Yaskawa INFORM job: test_long_tjr2.JBI

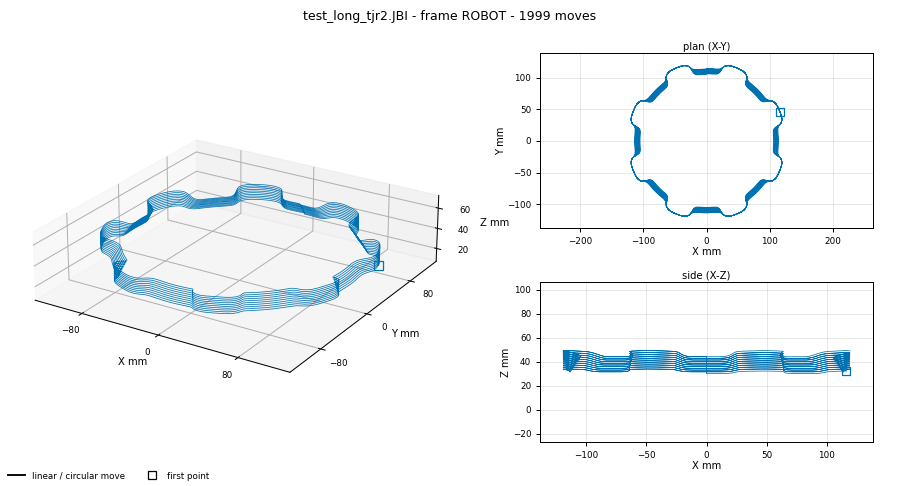
[picture p0: tool path of test_long_tjr2.JBI in frame ROBOT, 1999 of 2000 moves have a stored position in this frame; points joined in program order, loops and branches not executed]
version: 0
/JOB
//NAME test_long
//POS
///NPOS 48,0,0,2,0,0
///TOOL 1
///POSTYPE ROBOT
///RECTAN
///RCONF 1,0,0,0,0,0,0,0,0,0,0,0,0,0,0,0,0,0,0,0,0,0,0,0
C00000=117.720,41.900,32.250,-0.0000,-0.0000,1.0000
C00001=116.270,45.890,32.290,-0.0000,-0.0000,1.0000
C00002=114.660,49.770,32.290,-0.0000,-0.0000,1.0000
C00003=112.870,53.610,32.250,-0.0000,-0.0000,1.0000
C00004=110.690,57.360,32.180,0.0000,0.0000,1.0000
C00005=107.960,60.560,32.120,-0.0100,-0.0100,1.0000
C00006=105.150,62.790,32.030,-0.0300,-0.0400,1.0000
C00007=102.630,63.800,31.880,-0.0200,-0.0800,1.0000
C00008=100.220,64.240,31.550,-0.0200,-0.1500,0.9900
C00009=97.890,64.720,31.120,-0.0600,-0.2600,0.9600
C00010=95.560,65.770,30.680,-0.2000,-0.3600,0.9100
C00011=92.870,68.060,30.360,-0.3500,-0.3500,0.8700
C00012=89.340,72.130,30.220,-0.4000,-0.3400,0.8500
C00013=85.510,76.590,30.220,-0.3900,-0.3500,0.8500
C00014=81.180,81.180,30.220,-0.3700,-0.3700,0.8500
C00015=76.590,85.510,30.220,-0.3500,-0.3900,0.8500
C00016=72.130,89.340,30.220,-0.3400,-0.4000,0.8500
C00017=68.060,92.870,30.360,-0.3500,-0.3500,0.8700
C00018=65.770,95.560,30.680,-0.3600,-0.2000,0.9100
C00019=64.720,97.890,31.120,-0.2600,-0.0600,0.9600
C00020=64.240,100.220,31.550,-0.1500,-0.0200,0.9900
C00021=63.800,102.630,31.880,-0.0800,-0.0200,1.0000
C00022=62.790,105.150,32.030,-0.0400,-0.0300,1.0000
C00023=60.560,107.960,32.120,-0.0100,-0.0100,1.0000
C00024=57.360,110.690,32.180,0.0000,0.0000,1.0000
C00025=53.610,112.870,32.250,-0.0000,-0.0000,1.0000
C00026=49.770,114.660,32.290,-0.0000,-0.0000,1.0000
C00027=45.890,116.270,32.290,-0.0000,-0.0000,1.0000
C00028=41.900,117.720,32.250,-0.0000,-0.0000,1.0000
C00029=37.710,118.830,32.180,0.0000,0.0000,1.0000
C00030=33.520,119.170,32.120,0.0000,-0.0200,1.0000
C00031=29.950,118.750,32.030,0.0100,-0.0500,1.0000
C00032=27.450,117.680,31.880,0.0400,-0.0700,1.0000
C00033=25.440,116.290,31.550,0.0900,-0.1200,0.9900
C00034=23.450,114.980,31.120,0.1400,-0.2300,0.9600
C00035=21.060,114.080,30.680,0.1200,-0.3900,0.9100
C00036=17.540,113.790,30.360,0.0000,-0.5000,0.8700
C00037=12.170,114.170,30.220,-0.0400,-0.5200,0.8500
C00038=6.310,114.630,30.220,-0.0300,-0.5200,0.8500
C00039=0.000,114.800,30.220,0.0000,-0.5200,0.8500
C00040=0.000,113.910,31.670,0.0000,-0.5300,0.8500
C00041=6.230,113.730,31.660,-0.0300,-0.5300,0.8500
C00042=12.030,113.290,31.670,-0.0400,-0.5300,0.8500
C00043=17.380,112.940,31.810,0.0100,-0.5100,0.8600
C00044=20.850,113.300,32.180,0.1400,-0.3900,0.9100
C00045=23.220,114.320,32.670,0.1500,-0.2100,0.9700
C00046=25.180,115.780,33.150,0.0900,-0.1000,0.9900
C00047=27.170,117.350,33.520,0.0400,-0.0600,1.0000
C00048=29.650,118.590,33.700,0.0100,-0.0400,1.0000
C00049=33.230,119.130,33.790,0.0000,-0.0100,1.0000
C00050=37.480,118.870,33.870,0.0000,0.0000,1.0000
C00051=41.760,117.760,33.940,-0.0000,-0.0000,1.0000
C00052=45.840,116.290,33.990,-0.0000,-0.0000,1.0000
C00053=49.810,114.640,33.990,-0.0000,-0.0000,1.0000
C00054=53.740,112.800,33.940,-0.0000,-0.0000,1.0000
C00055=57.550,110.560,33.870,0.0000,0.0000,1.0000
C00056=60.740,107.740,33.790,-0.0100,-0.0100,1.0000
C00057=62.890,104.820,33.700,-0.0400,-0.0200,1.0000
C00058=63.760,102.190,33.520,-0.0700,-0.0100,1.0000
C00059=64.070,99.670,33.150,-0.1300,-0.0100,0.9900
C00060=64.420,97.260,32.670,-0.2500,-0.0500,0.9700
C00061=65.370,94.860,32.180,-0.3700,-0.1800,0.9100
C00062=67.570,92.150,31.810,-0.3700,-0.3500,0.8600
C00063=71.600,88.610,31.670,-0.3400,-0.4100,0.8500
C00064=76.020,84.820,31.660,-0.3600,-0.4000,0.8500
C00065=80.540,80.540,31.670,-0.3800,-0.3800,0.8500
C00066=84.820,76.020,31.660,-0.4000,-0.3600,0.8500
C00067=88.610,71.600,31.670,-0.4100,-0.3400,0.8500
C00068=92.150,67.570,31.810,-0.3500,-0.3700,0.8600
C00069=94.860,65.370,32.180,-0.1800,-0.3700,0.9100
C00070=97.260,64.420,32.670,-0.0500,-0.2500,0.9700
C00071=99.670,64.070,33.150,-0.0100,-0.1300,0.9900
C00072=102.190,63.760,33.520,-0.0100,-0.0700,1.0000
C00073=104.820,62.890,33.700,-0.0200,-0.0400,1.0000
C00074=107.740,60.740,33.790,-0.0100,-0.0100,1.0000
C00075=110.560,57.550,33.870,0.0000,0.0000,1.0000
C00076=112.800,53.740,33.940,-0.0000,-0.0000,1.0000
C00077=114.640,49.810,33.990,-0.0000,-0.0000,1.0000
C00078=116.290,45.840,33.990,-0.0000,-0.0000,1.0000
C00079=117.760,41.760,33.940,-0.0000,-0.0000,1.0000
C00080=118.870,37.480,33.870,0.0000,0.0000,1.0000
C00081=119.130,33.230,33.790,-0.0100,0.0000,1.0000
C00082=118.590,29.650,33.700,-0.0400,0.0100,1.0000
C00083=117.350,27.170,33.520,-0.0600,0.0400,1.0000
C00084=115.780,25.180,33.150,-0.1000,0.0900,0.9900
C00085=114.320,23.220,32.670,-0.2100,0.1500,0.9700
C00086=113.300,20.850,32.180,-0.3900,0.1400,0.9100
C00087=112.940,17.380,31.810,-0.5100,0.0100,0.8600
C00088=113.290,12.030,31.670,-0.5300,-0.0400,0.8500
C00089=113.730,6.230,31.660,-0.5300,-0.0300,0.8500
C00090=113.910,0.000,31.670,-0.5300,0.0000,0.8500
C00091=113.730,-6.230,31.660,-0.5300,0.0300,0.8500
C00092=113.290,-12.030,31.670,-0.5300,0.0400,0.8500
C00093=112.940,-17.380,31.810,-0.5100,-0.0100,0.8600
C00094=113.300,-20.850,32.180,-0.3900,-0.1400,0.9100
C00095=114.320,-23.220,32.670,-0.2100,-0.1500,0.9700
C00096=115.780,-25.180,33.150,-0.1000,-0.0900,0.9900
C00097=117.350,-27.170,33.520,-0.0600,-0.0400,1.0000
C00098=118.590,-29.650,33.700,-0.0400,-0.0100,1.0000
C00099=119.130,-33.230,33.790,-0.0100,-0.0000,1.0000
C00100=118.870,-37.480,33.870,0.0000,-0.0000,1.0000
C00101=117.760,-41.760,33.940,-0.0000,0.0000,1.0000
C00102=116.290,-45.840,33.990,-0.0000,0.0000,1.0000
C00103=114.640,-49.810,33.990,-0.0000,0.0000,1.0000
C00104=112.800,-53.740,33.940,-0.0000,0.0000,1.0000
C00105=110.560,-57.550,33.870,0.0000,-0.0000,1.0000
C00106=107.740,-60.740,33.790,-0.0100,0.0100,1.0000
C00107=104.820,-62.890,33.700,-0.0200,0.0400,1.0000
C00108=102.190,-63.760,33.520,-0.0100,0.0700,1.0000
C00109=99.670,-64.070,33.150,-0.0100,0.1300,0.9900
C00110=97.260,-64.420,32.670,-0.0500,0.2500,0.9700
C00111=94.860,-65.370,32.180,-0.1800,0.3700,0.9100
C00112=92.150,-67.570,31.810,-0.3500,0.3700,0.8600
C00113=88.610,-71.600,31.670,-0.4100,0.3400,0.8500
C00114=84.820,-76.020,31.660,-0.4000,0.3600,0.8500
C00115=80.540,-80.540,31.670,-0.3800,0.3800,0.8500
C00116=76.020,-84.820,31.660,-0.3600,0.4000,0.8500
C00117=71.600,-88.610,31.670,-0.3400,0.4100,0.8500
C00118=67.570,-92.150,31.810,-0.3700,0.3500,0.8600
C00119=65.370,-94.860,32.180,-0.3700,0.1800,0.9100
C00120=64.420,-97.260,32.670,-0.2500,0.0500,0.9700
C00121=64.070,-99.670,33.150,-0.1300,0.0100,0.9900
C00122=63.760,-102.190,33.520,-0.0700,0.0100,1.0000
C00123=62.890,-104.820,33.700,-0.0400,0.0200,1.0000
C00124=60.740,-107.740,33.790,-0.0100,0.0100,1.0000
C00125=57.550,-110.560,33.870,0.0000,-0.0000,1.0000
C00126=53.740,-112.800,33.940,-0.0000,0.0000,1.0000
C00127=49.810,-114.640,33.990,-0.0000,0.0000,1.0000
C00128=45.840,-116.290,33.990,-0.0000,0.0000,1.0000
C00129=41.760,-117.760,33.940,-0.0000,0.0000,1.0000
C00130=37.480,-118.870,33.870,0.0000,-0.0000,1.0000
C00131=33.230,-119.130,33.790,0.0000,0.0100,1.0000
C00132=29.650,-118.590,33.700,0.0100,0.0400,1.0000
C00133=27.170,-117.350,33.520,0.0400,0.0600,1.0000
C00134=25.180,-115.780,33.150,0.0900,0.1000,0.9900
C00135=23.220,-114.320,32.670,0.1500,0.2100,0.9700
C00136=20.850,-113.300,32.180,0.1400,0.3900,0.9100
C00137=17.380,-112.940,31.810,0.0100,0.5100,0.8600
C00138=12.030,-113.290,31.670,-0.0400,0.5300,0.8500
C00139=6.230,-113.730,31.660,-0.0300,0.5300,0.8500
C00140=0.000,-113.910,31.670,0.0000,0.5300,0.8500
C00141=0.000,-113.910,31.670,0.0000,0.5300,0.8500
C00142=-6.230,-113.730,31.660,0.0300,0.5300,0.8500
C00143=-12.030,-113.290,31.670,0.0400,0.5300,0.8500
C00144=-17.380,-112.940,31.810,-0.0100,0.5100,0.8600
C00145=-20.850,-113.300,32.180,-0.1400,0.3900,0.9100
C00146=-23.220,-114.320,32.670,-0.1500,0.2100,0.9700
C00147=-25.180,-115.780,33.150,-0.0900,0.1000,0.9900
C00148=-27.170,-117.350,33.520,-0.0400,0.0600,1.0000
C00149=-29.650,-118.590,33.700,-0.0100,0.0400,1.0000
C00150=-33.230,-119.130,33.790,-0.0000,0.0100,1.0000
C00151=-37.480,-118.870,33.870,-0.0000,-0.0000,1.0000
C00152=-41.760,-117.760,33.940,0.0000,0.0000,1.0000
C00153=-45.840,-116.290,33.990,0.0000,0.0000,1.0000
C00154=-49.810,-114.640,33.990,0.0000,0.0000,1.0000
C00155=-53.740,-112.800,33.940,0.0000,0.0000,1.0000
C00156=-57.550,-110.560,33.870,-0.0000,-0.0000,1.0000
C00157=-60.740,-107.740,33.790,0.0100,0.0100,1.0000
C00158=-62.890,-104.820,33.700,0.0400,0.0200,1.0000
C00159=-63.760,-102.190,33.520,0.0700,0.0100,1.0000
C00160=-64.070,-99.670,33.150,0.1300,0.0100,0.9900
C00161=-64.420,-97.260,32.670,0.2500,0.0500,0.9700
C00162=-65.370,-94.860,32.180,0.3700,0.1800,0.9100
C00163=-67.570,-92.150,31.810,0.3700,0.3500,0.8600
C00164=-71.600,-88.610,31.670,0.3400,0.4100,0.8500
C00165=-76.020,-84.820,31.660,0.3600,0.4000,0.8500
C00166=-80.540,-80.540,31.670,0.3800,0.3800,0.8500
C00167=-84.820,-76.020,31.660,0.4000,0.3600,0.8500
C00168=-88.610,-71.600,31.670,0.4100,0.3400,0.8500
C00169=-92.150,-67.570,31.810,0.3500,0.3700,0.8600
C00170=-94.860,-65.370,32.180,0.1800,0.3700,0.9100
C00171=-97.260,-64.420,32.670,0.0500,0.2500,0.9700
C00172=-99.670,-64.070,33.150,0.0100,0.1300,0.9900
C00173=-102.190,-63.760,33.520,0.0100,0.0700,1.0000
C00174=-104.820,-62.890,33.700,0.0200,0.0400,1.0000
C00175=-107.740,-60.740,33.790,0.0100,0.0100,1.0000
C00176=-110.560,-57.550,33.870,-0.0000,-0.0000,1.0000
C00177=-112.800,-53.740,33.940,0.0000,0.0000,1.0000
C00178=-114.640,-49.810,33.990,0.0000,0.0000,1.0000
C00179=-116.290,-45.840,33.990,0.0000,0.0000,1.0000
C00180=-117.760,-41.760,33.940,0.0000,0.0000,1.0000
C00181=-118.870,-37.480,33.870,-0.0000,-0.0000,1.0000
C00182=-119.130,-33.230,33.790,0.0100,-0.0000,1.0000
C00183=-118.590,-29.650,33.700,0.0400,-0.0100,1.0000
C00184=-117.350,-27.170,33.520,0.0600,-0.0400,1.0000
C00185=-115.780,-25.180,33.150,0.1000,-0.0900,0.9900
C00186=-114.320,-23.220,32.670,0.2100,-0.1500,0.9700
C00187=-113.300,-20.850,32.180,0.3900,-0.1400,0.9100
C00188=-112.940,-17.380,31.810,0.5100,-0.0100,0.8600
C00189=-113.290,-12.030,31.670,0.5300,0.0400,0.8500
C00190=-113.730,-6.230,31.660,0.5300,0.0300,0.8500
C00191=-113.910,0.000,31.670,0.5300,-0.0000,0.8500
C00192=-113.730,6.230,31.660,0.5300,-0.0300,0.8500
C00193=-113.290,12.030,31.670,0.5300,-0.0400,0.8500
C00194=-112.940,17.380,31.810,0.5100,0.0100,0.8600
C00195=-113.300,20.850,32.180,0.3900,0.1400,0.9100
C00196=-114.320,23.220,32.670,0.2100,0.1500,0.9700
C00197=-115.780,25.180,33.150,0.1000,0.0900,0.9900
C00198=-117.350,27.170,33.520,0.0600,0.0400,1.0000
C00199=-118.590,29.650,33.700,0.0400,0.0100,1.0000
C00200=-119.130,33.230,33.790,0.0100,0.0000,1.0000
C00201=-118.870,37.480,33.870,-0.0000,0.0000,1.0000
C00202=-117.760,41.760,33.940,0.0000,-0.0000,1.0000
C00203=-116.290,45.840,33.990,0.0000,-0.0000,1.0000
C00204=-114.640,49.810,33.990,0.0000,-0.0000,1.0000
C00205=-112.800,53.740,33.940,0.0000,-0.0000,1.0000
C00206=-110.560,57.550,33.870,-0.0000,0.0000,1.0000
C00207=-107.740,60.740,33.790,0.0100,-0.0100,1.0000
C00208=-104.820,62.890,33.700,0.0200,-0.0400,1.0000
C00209=-102.190,63.760,33.520,0.0100,-0.0700,1.0000
C00210=-99.670,64.070,33.150,0.0100,-0.1300,0.9900
C00211=-97.260,64.420,32.670,0.0500,-0.2500,0.9700
C00212=-94.860,65.370,32.180,0.1800,-0.3700,0.9100
C00213=-92.150,67.570,31.810,0.3500,-0.3700,0.8600
C00214=-88.610,71.600,31.670,0.4100,-0.3400,0.8500
C00215=-84.820,76.020,31.660,0.4000,-0.3600,0.8500
C00216=-80.540,80.540,31.670,0.3800,-0.3800,0.8500
C00217=-76.020,84.820,31.660,0.3600,-0.4000,0.8500
C00218=-71.600,88.610,31.670,0.3400,-0.4100,0.8500
C00219=-67.570,92.150,31.810,0.3700,-0.3500,0.8600
C00220=-65.370,94.860,32.180,0.3700,-0.1800,0.9100
C00221=-64.420,97.260,32.670,0.2500,-0.0500,0.9700
C00222=-64.070,99.670,33.150,0.1300,-0.0100,0.9900
C00223=-63.760,102.190,33.520,0.0700,-0.0100,1.0000
C00224=-62.890,104.820,33.700,0.0400,-0.0200,1.0000
C00225=-60.740,107.740,33.790,0.0100,-0.0100,1.0000
C00226=-57.550,110.560,33.870,-0.0000,0.0000,1.0000
C00227=-53.740,112.800,33.940,0.0000,-0.0000,1.0000
C00228=-49.810,114.640,33.990,0.0000,-0.0000,1.0000
C00229=-45.840,116.290,33.990,0.0000,-0.0000,1.0000
C00230=-41.760,117.760,33.940,0.0000,-0.0000,1.0000
C00231=-37.480,118.870,33.870,-0.0000,0.0000,1.0000
C00232=-33.230,119.130,33.790,-0.0000,-0.0100,1.0000
C00233=-29.650,118.590,33.700,-0.0100,-0.0400,1.0000
C00234=-27.170,117.350,33.520,-0.0400,-0.0600,1.0000
C00235=-25.180,115.780,33.150,-0.0900,-0.1000,0.9900
C00236=-23.220,114.320,32.670,-0.1500,-0.2100,0.9700
C00237=-20.850,113.300,32.180,-0.1400,-0.3900,0.9100
C00238=-17.380,112.940,31.810,-0.0100,-0.5100,0.8600
C00239=-12.030,113.290,31.670,0.0400,-0.5300,0.8500
C00240=-6.230,113.730,31.660,0.0300,-0.5300,0.8500
C00241=0.000,113.910,31.670,0.0000,-0.5300,0.8500
C00242=0.000,112.990,33.100,0.0000,-0.5400,0.8400
C00243=-6.140,112.820,33.090,0.0300,-0.5400,0.8400
C00244=-11.890,112.380,33.100,0.0400,-0.5400,0.8400
C00245=-17.200,112.060,33.260,-0.0200,-0.5200,0.8500
C00246=-20.640,112.500,33.660,-0.1500,-0.3800,0.9100
C00247=-22.970,113.650,34.210,-0.1500,-0.1900,0.9700
C00248=-24.910,115.260,34.750,-0.0800,-0.0900,0.9900
C00249=-26.890,117.010,35.160,-0.0300,-0.0400,1.0000
C00250=-29.330,118.420,35.360,-0.0100,-0.0300,1.0000
C00251=-32.930,119.100,35.460,-0.0000,-0.0100,1.0000
C00252=-37.250,118.910,35.550,-0.0000,0.0100,1.0000
C00253=-41.610,117.810,35.640,0.0000,-0.0000,1.0000
C00254=-45.790,116.310,35.690,0.0000,-0.0000,1.0000
C00255=-49.860,114.620,35.690,0.0000,-0.0000,1.0000
C00256=-53.880,112.730,35.640,0.0000,-0.0000,1.0000
C00257=-57.740,110.420,35.550,-0.0000,0.0000,1.0000
C00258=-60.930,107.500,35.460,0.0100,-0.0100,1.0000
C00259=-62.990,104.470,35.360,0.0300,-0.0100,1.0000
C00260=-63.730,101.750,35.160,0.0600,-0.0100,1.0000
C00261=-63.890,99.120,34.750,0.1200,-0.0000,0.9900
C00262=-64.120,96.610,34.210,0.2400,-0.0300,0.9700
C00263=-64.960,94.150,33.660,0.3800,-0.1600,0.9100
C00264=-67.080,91.410,33.260,0.3800,-0.3500,0.8500
C00265=-71.060,87.870,33.100,0.3500,-0.4100,0.8400
C00266=-75.430,84.120,33.090,0.3600,-0.4100,0.8400
C00267=-79.900,79.900,33.100,0.3800,-0.3800,0.8400
C00268=-84.120,75.430,33.090,0.4100,-0.3600,0.8400
C00269=-87.870,71.060,33.100,0.4100,-0.3500,0.8400
C00270=-91.410,67.080,33.260,0.3500,-0.3800,0.8500
C00271=-94.150,64.960,33.660,0.1600,-0.3800,0.9100
C00272=-96.610,64.120,34.210,0.0300,-0.2400,0.9700
C00273=-99.120,63.890,34.750,0.0000,-0.1200,0.9900
C00274=-101.750,63.730,35.160,0.0100,-0.0600,1.0000
C00275=-104.470,62.990,35.360,0.0100,-0.0300,1.0000
C00276=-107.500,60.930,35.460,0.0100,-0.0100,1.0000
C00277=-110.420,57.740,35.550,-0.0000,0.0000,1.0000
C00278=-112.730,53.880,35.640,0.0000,-0.0000,1.0000
C00279=-114.620,49.860,35.690,0.0000,-0.0000,1.0000
C00280=-116.310,45.790,35.690,0.0000,-0.0000,1.0000
C00281=-117.810,41.610,35.640,0.0000,-0.0000,1.0000
C00282=-118.910,37.250,35.550,-0.0100,0.0000,1.0000
C00283=-119.100,32.930,35.460,0.0100,0.0000,1.0000
C00284=-118.420,29.330,35.360,0.0300,0.0100,1.0000
C00285=-117.010,26.890,35.160,0.0400,0.0300,1.0000
C00286=-115.260,24.910,34.750,0.0900,0.0800,0.9900
C00287=-113.650,22.970,34.210,0.1900,0.1500,0.9700
C00288=-112.500,20.640,33.660,0.3800,0.1500,0.9100
C00289=-112.060,17.200,33.260,0.5200,0.0200,0.8500
C00290=-112.380,11.890,33.100,0.5400,-0.0400,0.8400
C00291=-112.820,6.140,33.090,0.5400,-0.0300,0.8400
C00292=-112.990,0.000,33.100,0.5400,-0.0000,0.8400
C00293=-112.820,-6.140,33.090,0.5400,0.0300,0.8400
C00294=-112.380,-11.890,33.100,0.5400,0.0400,0.8400
C00295=-112.060,-17.200,33.260,0.5200,-0.0200,0.8500
C00296=-112.500,-20.640,33.660,0.3800,-0.1500,0.9100
C00297=-113.650,-22.970,34.210,0.1900,-0.1500,0.9700
C00298=-115.260,-24.910,34.750,0.0900,-0.0800,0.9900
C00299=-117.010,-26.890,35.160,0.0400,-0.0300,1.0000
C00300=-118.420,-29.330,35.360,0.0300,-0.0100,1.0000
C00301=-119.100,-32.930,35.460,0.0100,-0.0000,1.0000
C00302=-118.910,-37.250,35.550,-0.0100,-0.0000,1.0000
C00303=-117.810,-41.610,35.640,0.0000,0.0000,1.0000
C00304=-116.310,-45.790,35.690,0.0000,0.0000,1.0000
C00305=-114.620,-49.860,35.690,0.0000,0.0000,1.0000
C00306=-112.730,-53.880,35.640,0.0000,0.0000,1.0000
C00307=-110.420,-57.740,35.550,-0.0000,-0.0000,1.0000
C00308=-107.500,-60.930,35.460,0.0100,0.0100,1.0000
C00309=-104.470,-62.990,35.360,0.0100,0.0300,1.0000
C00310=-101.750,-63.730,35.160,0.0100,0.0600,1.0000
C00311=-99.120,-63.890,34.750,0.0000,0.1200,0.9900
C00312=-96.610,-64.120,34.210,0.0300,0.2400,0.9700
C00313=-94.150,-64.960,33.660,0.1600,0.3800,0.9100
C00314=-91.410,-67.080,33.260,0.3500,0.3800,0.8500
C00315=-87.870,-71.060,33.100,0.4100,0.3500,0.8400
C00316=-84.120,-75.430,33.090,0.4100,0.3600,0.8400
C00317=-79.900,-79.900,33.100,0.3800,0.3800,0.8400
C00318=-75.430,-84.120,33.090,0.3600,0.4100,0.8400
C00319=-71.060,-87.870,33.100,0.3500,0.4100,0.8400
C00320=-67.080,-91.410,33.260,0.3800,0.3500,0.8500
C00321=-64.960,-94.150,33.660,0.3800,0.1600,0.9100
C00322=-64.120,-96.610,34.210,0.2400,0.0300,0.9700
C00323=-63.890,-99.120,34.750,0.1200,0.0000,0.9900
C00324=-63.730,-101.750,35.160,0.0600,0.0100,1.0000
C00325=-62.990,-104.470,35.360,0.0300,0.0100,1.0000
C00326=-60.930,-107.500,35.460,0.0100,0.0100,1.0000
C00327=-57.740,-110.420,35.550,-0.0000,-0.0000,1.0000
C00328=-53.880,-112.730,35.640,0.0000,0.0000,1.0000
C00329=-49.860,-114.620,35.690,0.0000,0.0000,1.0000
C00330=-45.790,-116.310,35.690,0.0000,0.0000,1.0000
C00331=-41.610,-117.810,35.640,0.0000,0.0000,1.0000
C00332=-37.250,-118.910,35.550,-0.0000,-0.0100,1.0000
C00333=-32.930,-119.100,35.460,-0.0000,0.0100,1.0000
C00334=-29.330,-118.420,35.360,-0.0100,0.0300,1.0000
C00335=-26.890,-117.010,35.160,-0.0300,0.0400,1.0000
C00336=-24.910,-115.260,34.750,-0.0800,0.0900,0.9900
C00337=-22.970,-113.650,34.210,-0.1500,0.1900,0.9700
C00338=-20.640,-112.500,33.660,-0.1500,0.3800,0.9100
C00339=-17.200,-112.060,33.260,-0.0200,0.5200,0.8500
C00340=-11.890,-112.380,33.100,0.0400,0.5400,0.8400
C00341=-6.140,-112.820,33.090,0.0300,0.5400,0.8400
C00342=0.000,-112.990,33.100,0.0000,0.5400,0.8400
C00343=0.000,-112.990,33.100,0.0000,0.5400,0.8400
C00344=6.140,-112.820,33.090,-0.0300,0.5400,0.8400
C00345=11.890,-112.380,33.100,-0.0400,0.5400,0.8400
C00346=17.200,-112.060,33.260,0.0200,0.5200,0.8500
C00347=20.640,-112.500,33.660,0.1500,0.3800,0.9100
C00348=22.970,-113.650,34.210,0.1500,0.1900,0.9700
C00349=24.910,-115.260,34.750,0.0800,0.0900,0.9900
C00350=26.890,-117.010,35.160,0.0300,0.0400,1.0000
C00351=29.330,-118.420,35.360,0.0100,0.0300,1.0000
C00352=32.930,-119.100,35.460,0.0000,0.0100,1.0000
C00353=37.250,-118.910,35.550,0.0000,-0.0100,1.0000
C00354=41.610,-117.810,35.640,-0.0000,0.0000,1.0000
C00355=45.790,-116.310,35.690,-0.0000,0.0000,1.0000
C00356=49.860,-114.620,35.690,-0.0000,0.0000,1.0000
C00357=53.880,-112.730,35.640,-0.0000,0.0000,1.0000
C00358=57.740,-110.420,35.550,0.0000,-0.0000,1.0000
C00359=60.930,-107.500,35.460,-0.0100,0.0100,1.0000
C00360=62.990,-104.470,35.360,-0.0300,0.0100,1.0000
C00361=63.730,-101.750,35.160,-0.0600,0.0100,1.0000
C00362=63.890,-99.120,34.750,-0.1200,0.0000,0.9900
C00363=64.120,-96.610,34.210,-0.2400,0.0300,0.9700
C00364=64.960,-94.150,33.660,-0.3800,0.1600,0.9100
C00365=67.080,-91.410,33.260,-0.3800,0.3500,0.8500
C00366=71.060,-87.870,33.100,-0.3500,0.4100,0.8400
C00367=75.430,-84.120,33.090,-0.3600,0.4100,0.8400
C00368=79.900,-79.900,33.100,-0.3800,0.3800,0.8400
C00369=84.120,-75.430,33.090,-0.4100,0.3600,0.8400
C00370=87.870,-71.060,33.100,-0.4100,0.3500,0.8400
C00371=91.410,-67.080,33.260,-0.3500,0.3800,0.8500
C00372=94.150,-64.960,33.660,-0.1600,0.3800,0.9100
C00373=96.610,-64.120,34.210,-0.0300,0.2400,0.9700
C00374=99.120,-63.890,34.750,-0.0000,0.1200,0.9900
C00375=101.750,-63.730,35.160,-0.0100,0.0600,1.0000
C00376=104.470,-62.990,35.360,-0.0100,0.0300,1.0000
C00377=107.500,-60.930,35.460,-0.0100,0.0100,1.0000
C00378=110.420,-57.740,35.550,0.0000,-0.0000,1.0000
C00379=112.730,-53.880,35.640,-0.0000,0.0000,1.0000
C00380=114.620,-49.860,35.690,-0.0000,0.0000,1.0000
C00381=116.310,-45.790,35.690,-0.0000,0.0000,1.0000
C00382=117.810,-41.610,35.640,-0.0000,0.0000,1.0000
C00383=118.910,-37.250,35.550,0.0100,-0.0000,1.0000
C00384=119.100,-32.930,35.460,-0.0100,-0.0000,1.0000
C00385=118.420,-29.330,35.360,-0.0300,-0.0100,1.0000
C00386=117.010,-26.890,35.160,-0.0400,-0.0300,1.0000
C00387=115.260,-24.910,34.750,-0.0900,-0.0800,0.9900
C00388=113.650,-22.970,34.210,-0.1900,-0.1500,0.9700
C00389=112.500,-20.640,33.660,-0.3800,-0.1500,0.9100
C00390=112.060,-17.200,33.260,-0.5200,-0.0200,0.8500
C00391=112.380,-11.890,33.100,-0.5400,0.0400,0.8400
C00392=112.820,-6.140,33.090,-0.5400,0.0300,0.8400
C00393=112.990,0.000,33.100,-0.5400,0.0000,0.8400
C00394=112.820,6.140,33.090,-0.5400,-0.0300,0.8400
C00395=112.380,11.890,33.100,-0.5400,-0.0400,0.8400
C00396=112.060,17.200,33.260,-0.5200,0.0200,0.8500
C00397=112.500,20.640,33.660,-0.3800,0.1500,0.9100
C00398=113.650,22.970,34.210,-0.1900,0.1500,0.9700
C00399=115.260,24.910,34.750,-0.0900,0.0800,0.9900
C00400=117.010,26.890,35.160,-0.0400,0.0300,1.0000
C00401=118.420,29.330,35.360,-0.0300,0.0100,1.0000
C00402=119.100,32.930,35.460,-0.0100,0.0000,1.0000
C00403=118.910,37.250,35.550,0.0100,0.0000,1.0000
C00404=117.810,41.610,35.640,-0.0000,-0.0000,1.0000
C00405=116.310,45.790,35.690,-0.0000,-0.0000,1.0000
C00406=114.620,49.860,35.690,-0.0000,-0.0000,1.0000
C00407=112.730,53.880,35.640,-0.0000,-0.0000,1.0000
C00408=110.420,57.740,35.550,0.0000,0.0000,1.0000
C00409=107.500,60.930,35.460,-0.0100,-0.0100,1.0000
C00410=104.470,62.990,35.360,-0.0100,-0.0300,1.0000
C00411=101.750,63.730,35.160,-0.0100,-0.0600,1.0000
C00412=99.120,63.890,34.750,-0.0000,-0.1200,0.9900
C00413=96.610,64.120,34.210,-0.0300,-0.2400,0.9700
C00414=94.150,64.960,33.660,-0.1600,-0.3800,0.9100
C00415=91.410,67.080,33.260,-0.3500,-0.3800,0.8500
C00416=87.870,71.060,33.100,-0.4100,-0.3500,0.8400
C00417=84.120,75.430,33.090,-0.4100,-0.3600,0.8400
C00418=79.900,79.900,33.100,-0.3800,-0.3800,0.8400
C00419=75.430,84.120,33.090,-0.3600,-0.4100,0.8400
C00420=71.060,87.870,33.100,-0.3500,-0.4100,0.8400
C00421=67.080,91.410,33.260,-0.3800,-0.3500,0.8500
C00422=64.960,94.150,33.660,-0.3800,-0.1600,0.9100
C00423=64.120,96.610,34.210,-0.2400,-0.0300,0.9700
C00424=63.890,99.120,34.750,-0.1200,-0.0000,0.9900
C00425=63.730,101.750,35.160,-0.0600,-0.0100,1.0000
C00426=62.990,104.470,35.360,-0.0300,-0.0100,1.0000
C00427=60.930,107.500,35.460,-0.0100,-0.0100,1.0000
C00428=57.740,110.420,35.550,0.0000,0.0000,1.0000
C00429=53.880,112.730,35.640,-0.0000,-0.0000,1.0000
C00430=49.860,114.620,35.690,-0.0000,-0.0000,1.0000
C00431=45.790,116.310,35.690,-0.0000,-0.0000,1.0000
C00432=41.610,117.810,35.640,-0.0000,-0.0000,1.0000
C00433=37.250,118.910,35.550,0.0000,0.0100,1.0000
C00434=32.930,119.100,35.460,0.0000,-0.0100,1.0000
C00435=29.330,118.420,35.360,0.0100,-0.0300,1.0000
C00436=26.890,117.010,35.160,0.0300,-0.0400,1.0000
C00437=24.910,115.260,34.750,0.0800,-0.0900,0.9900
C00438=22.970,113.650,34.210,0.1500,-0.1900,0.9700
C00439=20.640,112.500,33.660,0.1500,-0.3800,0.9100
C00440=17.200,112.060,33.260,0.0200,-0.5200,0.8500
C00441=11.890,112.380,33.100,-0.0400,-0.5400,0.8400
C00442=6.140,112.820,33.090,-0.0300,-0.5400,0.8400
C00443=0.000,112.990,33.100,0.0000,-0.5400,0.8400
C00444=0.000,112.060,34.520,0.0000,-0.5500,0.8300
C00445=6.060,111.890,34.510,-0.0300,-0.5500,0.8300
C00446=11.750,111.460,34.520,-0.0400,-0.5500,0.8300
C00447=17.030,111.170,34.700,0.0300,-0.5300,0.8500
C00448=20.430,111.690,35.140,0.1700,-0.3700,0.9100
C00449=22.720,112.950,35.740,0.1500,-0.1700,0.9700
C00450=24.640,114.730,36.340,0.0800,-0.0700,0.9900
C00451=26.590,116.660,36.800,0.0300,-0.0300,1.0000
C00452=29.010,118.240,37.020,0.0100,-0.0200,1.0000
C00453=32.630,119.060,37.140,0.0000,-0.0100,1.0000
C00454=37.000,118.950,37.230,0.0000,0.0100,1.0000
C00455=41.460,117.860,37.330,-0.0000,-0.0000,1.0000
C00456=45.730,116.330,37.390,-0.0000,-0.0000,1.0000
C00457=49.920,114.590,37.390,-0.0000,-0.0000,1.0000
C00458=54.030,112.660,37.330,-0.0000,-0.0000,1.0000
C00459=57.950,110.280,37.230,0.0000,0.0100,1.0000
C00460=61.120,107.260,37.140,-0.0000,-0.0000,1.0000
C00461=63.100,104.120,37.020,-0.0200,-0.0100,1.0000
C00462=63.690,101.290,36.800,-0.0400,-0.0000,1.0000
C00463=63.700,98.550,36.340,-0.1000,0.0000,0.9900
C00464=63.800,95.940,35.740,-0.2300,-0.0200,0.9700
C00465=64.530,93.420,35.140,-0.3800,-0.1400,0.9100
C00466=66.570,90.650,34.700,-0.3900,-0.3500,0.8500
C00467=70.510,87.120,34.520,-0.3600,-0.4200,0.8300
C00468=74.830,83.400,34.510,-0.3700,-0.4100,0.8300
C00469=79.240,79.240,34.520,-0.3900,-0.3900,0.8300
C00470=83.400,74.830,34.510,-0.4100,-0.3700,0.8300
C00471=87.120,70.510,34.520,-0.4200,-0.3600,0.8300
C00472=90.650,66.570,34.700,-0.3500,-0.3900,0.8500
C00473=93.420,64.530,35.140,-0.1400,-0.3800,0.9100
C00474=95.940,63.800,35.740,-0.0200,-0.2300,0.9700
C00475=98.550,63.700,36.340,0.0000,-0.1000,0.9900
C00476=101.290,63.690,36.800,-0.0000,-0.0400,1.0000
C00477=104.120,63.100,37.020,-0.0100,-0.0200,1.0000
C00478=107.260,61.120,37.140,-0.0000,-0.0000,1.0000
C00479=110.280,57.950,37.230,0.0100,0.0000,1.0000
C00480=112.660,54.030,37.330,-0.0000,-0.0000,1.0000
C00481=114.590,49.920,37.390,-0.0000,-0.0000,1.0000
C00482=116.330,45.730,37.390,-0.0000,-0.0000,1.0000
C00483=117.860,41.460,37.330,-0.0000,-0.0000,1.0000
C00484=118.950,37.000,37.230,0.0100,0.0000,1.0000
C00485=119.060,32.630,37.140,-0.0100,0.0000,1.0000
C00486=118.240,29.010,37.020,-0.0200,0.0100,1.0000
C00487=116.660,26.590,36.800,-0.0300,0.0300,1.0000
C00488=114.730,24.640,36.340,-0.0700,0.0800,0.9900
C00489=112.950,22.720,35.740,-0.1700,0.1500,0.9700
C00490=111.690,20.430,35.140,-0.3700,0.1700,0.9100
C00491=111.170,17.030,34.700,-0.5300,0.0300,0.8500
C00492=111.460,11.750,34.520,-0.5500,-0.0400,0.8300
C00493=111.890,6.060,34.510,-0.5500,-0.0300,0.8300
C00494=112.060,0.000,34.520,-0.5500,0.0000,0.8300
C00495=111.890,-6.060,34.510,-0.5500,0.0300,0.8300
C00496=111.460,-11.750,34.520,-0.5500,0.0400,0.8300
C00497=111.170,-17.030,34.700,-0.5300,-0.0300,0.8500
C00498=111.690,-20.430,35.140,-0.3700,-0.1700,0.9100
C00499=112.950,-22.720,35.740,-0.1700,-0.1500,0.9700
C00500=114.730,-24.640,36.340,-0.0700,-0.0800,0.9900
C00501=116.660,-26.590,36.800,-0.0300,-0.0300,1.0000
C00502=118.240,-29.010,37.020,-0.0200,-0.0100,1.0000
C00503=119.060,-32.630,37.140,-0.0100,-0.0000,1.0000
C00504=118.950,-37.000,37.230,0.0100,-0.0000,1.0000
C00505=117.860,-41.460,37.330,-0.0000,0.0000,1.0000
C00506=116.330,-45.730,37.390,-0.0000,0.0000,1.0000
C00507=114.590,-49.920,37.390,-0.0000,0.0000,1.0000
C00508=112.660,-54.030,37.330,-0.0000,0.0000,1.0000
C00509=110.280,-57.950,37.230,0.0100,-0.0000,1.0000
C00510=107.260,-61.120,37.140,-0.0000,0.0000,1.0000
C00511=104.120,-63.100,37.020,-0.0100,0.0200,1.0000
C00512=101.290,-63.690,36.800,-0.0000,0.0400,1.0000
C00513=98.550,-63.700,36.340,0.0000,0.1000,0.9900
C00514=95.940,-63.800,35.740,-0.0200,0.2300,0.9700
C00515=93.420,-64.530,35.140,-0.1400,0.3800,0.9100
C00516=90.650,-66.570,34.700,-0.3500,0.3900,0.8500
C00517=87.120,-70.510,34.520,-0.4200,0.3600,0.8300
C00518=83.400,-74.830,34.510,-0.4100,0.3700,0.8300
C00519=79.240,-79.240,34.520,-0.3900,0.3900,0.8300
C00520=74.830,-83.400,34.510,-0.3700,0.4100,0.8300
C00521=70.510,-87.120,34.520,-0.3600,0.4200,0.8300
C00522=66.570,-90.650,34.700,-0.3900,0.3500,0.8500
C00523=64.530,-93.420,35.140,-0.3800,0.1400,0.9100
C00524=63.800,-95.940,35.740,-0.2300,0.0200,0.9700
C00525=63.700,-98.550,36.340,-0.1000,-0.0000,0.9900
C00526=63.690,-101.290,36.800,-0.0400,0.0000,1.0000
C00527=63.100,-104.120,37.020,-0.0200,0.0100,1.0000
C00528=61.120,-107.260,37.140,-0.0000,0.0000,1.0000
C00529=57.950,-110.280,37.230,0.0000,-0.0100,1.0000
C00530=54.030,-112.660,37.330,-0.0000,0.0000,1.0000
C00531=49.920,-114.590,37.390,-0.0000,0.0000,1.0000
C00532=45.730,-116.330,37.390,-0.0000,0.0000,1.0000
C00533=41.460,-117.860,37.330,-0.0000,0.0000,1.0000
C00534=37.000,-118.950,37.230,0.0000,-0.0100,1.0000
C00535=32.630,-119.060,37.140,0.0000,0.0100,1.0000
C00536=29.010,-118.240,37.020,0.0100,0.0200,1.0000
C00537=26.590,-116.660,36.800,0.0300,0.0300,1.0000
C00538=24.640,-114.730,36.340,0.0800,0.0700,0.9900
C00539=22.720,-112.950,35.740,0.1500,0.1700,0.9700
C00540=20.430,-111.690,35.140,0.1700,0.3700,0.9100
C00541=17.030,-111.170,34.700,0.0300,0.5300,0.8500
C00542=11.750,-111.460,34.520,-0.0400,0.5500,0.8300
C00543=6.060,-111.890,34.510,-0.0300,0.5500,0.8300
C00544=0.000,-112.060,34.520,0.0000,0.5500,0.8300
C00545=0.000,-112.060,34.520,0.0000,0.5500,0.8300
C00546=-6.060,-111.890,34.510,0.0300,0.5500,0.8300
C00547=-11.750,-111.460,34.520,0.0400,0.5500,0.8300
C00548=-17.030,-111.170,34.700,-0.0300,0.5300,0.8500
C00549=-20.430,-111.690,35.140,-0.1700,0.3700,0.9100
C00550=-22.720,-112.950,35.740,-0.1500,0.1700,0.9700
C00551=-24.640,-114.730,36.340,-0.0800,0.0700,0.9900
C00552=-26.590,-116.660,36.800,-0.0300,0.0300,1.0000
C00553=-29.010,-118.240,37.020,-0.0100,0.0200,1.0000
C00554=-32.630,-119.060,37.140,-0.0000,0.0100,1.0000
C00555=-37.000,-118.950,37.230,-0.0000,-0.0100,1.0000
C00556=-41.460,-117.860,37.330,0.0000,0.0000,1.0000
C00557=-45.730,-116.330,37.390,0.0000,0.0000,1.0000
C00558=-49.920,-114.590,37.390,0.0000,0.0000,1.0000
C00559=-54.030,-112.660,37.330,0.0000,0.0000,1.0000
C00560=-57.950,-110.280,37.230,-0.0000,-0.0100,1.0000
C00561=-61.120,-107.260,37.140,0.0000,0.0000,1.0000
C00562=-63.100,-104.120,37.020,0.0200,0.0100,1.0000
C00563=-63.690,-101.290,36.800,0.0400,0.0000,1.0000
C00564=-63.700,-98.550,36.340,0.1000,-0.0000,0.9900
C00565=-63.800,-95.940,35.740,0.2300,0.0200,0.9700
C00566=-64.530,-93.420,35.140,0.3800,0.1400,0.9100
C00567=-66.570,-90.650,34.700,0.3900,0.3500,0.8500
C00568=-70.510,-87.120,34.520,0.3600,0.4200,0.8300
C00569=-74.830,-83.400,34.510,0.3700,0.4100,0.8300
C00570=-79.240,-79.240,34.520,0.3900,0.3900,0.8300
C00571=-83.400,-74.830,34.510,0.4100,0.3700,0.8300
C00572=-87.120,-70.510,34.520,0.4200,0.3600,0.8300
C00573=-90.650,-66.570,34.700,0.3500,0.3900,0.8500
C00574=-93.420,-64.530,35.140,0.1400,0.3800,0.9100
C00575=-95.940,-63.800,35.740,0.0200,0.2300,0.9700
C00576=-98.550,-63.700,36.340,-0.0000,0.1000,0.9900
C00577=-101.290,-63.690,36.800,0.0000,0.0400,1.0000
C00578=-104.120,-63.100,37.020,0.0100,0.0200,1.0000
C00579=-107.260,-61.120,37.140,0.0000,0.0000,1.0000
C00580=-110.280,-57.950,37.230,-0.0100,-0.0000,1.0000
C00581=-112.660,-54.030,37.330,0.0000,0.0000,1.0000
C00582=-114.590,-49.920,37.390,0.0000,0.0000,1.0000
C00583=-116.330,-45.730,37.390,0.0000,0.0000,1.0000
C00584=-117.860,-41.460,37.330,0.0000,0.0000,1.0000
C00585=-118.950,-37.000,37.230,-0.0100,-0.0000,1.0000
C00586=-119.060,-32.630,37.140,0.0100,-0.0000,1.0000
C00587=-118.240,-29.010,37.020,0.0200,-0.0100,1.0000
C00588=-116.660,-26.590,36.800,0.0300,-0.0300,1.0000
C00589=-114.730,-24.640,36.340,0.0700,-0.0800,0.9900
C00590=-112.950,-22.720,35.740,0.1700,-0.1500,0.9700
C00591=-111.690,-20.430,35.140,0.3700,-0.1700,0.9100
C00592=-111.170,-17.030,34.700,0.5300,-0.0300,0.8500
C00593=-111.460,-11.750,34.520,0.5500,0.0400,0.8300
C00594=-111.890,-6.060,34.510,0.5500,0.0300,0.8300
C00595=-112.060,0.000,34.520,0.5500,-0.0000,0.8300
C00596=-111.890,6.060,34.510,0.5500,-0.0300,0.8300
C00597=-111.460,11.750,34.520,0.5500,-0.0400,0.8300
C00598=-111.170,17.030,34.700,0.5300,0.0300,0.8500
C00599=-111.690,20.430,35.140,0.3700,0.1700,0.9100
C00600=-112.950,22.720,35.740,0.1700,0.1500,0.9700
C00601=-114.730,24.640,36.340,0.0700,0.0800,0.9900
C00602=-116.660,26.590,36.800,0.0300,0.0300,1.0000
C00603=-118.240,29.010,37.020,0.0200,0.0100,1.0000
C00604=-119.060,32.630,37.140,0.0100,0.0000,1.0000
C00605=-118.950,37.000,37.230,-0.0100,0.0000,1.0000
C00606=-117.860,41.460,37.330,0.0000,-0.0000,1.0000
C00607=-116.330,45.730,37.390,0.0000,-0.0000,1.0000
C00608=-114.590,49.920,37.390,0.0000,-0.0000,1.0000
C00609=-112.660,54.030,37.330,0.0000,-0.0000,1.0000
C00610=-110.280,57.950,37.230,-0.0100,0.0000,1.0000
C00611=-107.260,61.120,37.140,0.0000,-0.0000,1.0000
C00612=-104.120,63.100,37.020,0.0100,-0.0200,1.0000
C00613=-101.290,63.690,36.800,0.0000,-0.0400,1.0000
C00614=-98.550,63.700,36.340,-0.0000,-0.1000,0.9900
C00615=-95.940,63.800,35.740,0.0200,-0.2300,0.9700
C00616=-93.420,64.530,35.140,0.1400,-0.3800,0.9100
C00617=-90.650,66.570,34.700,0.3500,-0.3900,0.8500
C00618=-87.120,70.510,34.520,0.4200,-0.3600,0.8300
C00619=-83.400,74.830,34.510,0.4100,-0.3700,0.8300
C00620=-79.240,79.240,34.520,0.3900,-0.3900,0.8300
C00621=-74.830,83.400,34.510,0.3700,-0.4100,0.8300
C00622=-70.510,87.120,34.520,0.3600,-0.4200,0.8300
C00623=-66.570,90.650,34.700,0.3900,-0.3500,0.8500
C00624=-64.530,93.420,35.140,0.3800,-0.1400,0.9100
C00625=-63.800,95.940,35.740,0.2300,-0.0200,0.9700
C00626=-63.700,98.550,36.340,0.1000,0.0000,0.9900
C00627=-63.690,101.290,36.800,0.0400,-0.0000,1.0000
C00628=-63.100,104.120,37.020,0.0200,-0.0100,1.0000
C00629=-61.120,107.260,37.140,0.0000,-0.0000,1.0000
C00630=-57.950,110.280,37.230,-0.0000,0.0100,1.0000
C00631=-54.030,112.660,37.330,0.0000,-0.0000,1.0000
C00632=-49.920,114.590,37.390,0.0000,-0.0000,1.0000
C00633=-45.730,116.330,37.390,0.0000,-0.0000,1.0000
C00634=-41.460,117.860,37.330,0.0000,-0.0000,1.0000
C00635=-37.000,118.950,37.230,-0.0000,0.0100,1.0000
C00636=-32.630,119.060,37.140,-0.0000,-0.0100,1.0000
C00637=-29.010,118.240,37.020,-0.0100,-0.0200,1.0000
C00638=-26.590,116.660,36.800,-0.0300,-0.0300,1.0000
C00639=-24.640,114.730,36.340,-0.0800,-0.0700,0.9900
C00640=-22.720,112.950,35.740,-0.1500,-0.1700,0.9700
C00641=-20.430,111.690,35.140,-0.1700,-0.3700,0.9100
C00642=-17.030,111.170,34.700,-0.0300,-0.5300,0.8500
C00643=-11.750,111.460,34.520,0.0400,-0.5500,0.8300
C00644=-6.060,111.890,34.510,0.0300,-0.5500,0.8300
C00645=0.000,112.060,34.520,0.0000,-0.5500,0.8300
C00646=0.000,111.100,35.930,0.0000,-0.5600,0.8300
C00647=-5.970,110.940,35.920,0.0300,-0.5600,0.8300
C00648=-11.600,110.520,35.930,0.0400,-0.5600,0.8300
C00649=-16.850,110.260,36.120,-0.0400,-0.5300,0.8400
C00650=-20.210,110.860,36.610,-0.1800,-0.3600,0.9200
C00651=-22.470,112.250,37.260,-0.1500,-0.1600,0.9800
C00652=-24.360,114.180,37.930,-0.0700,-0.0600,1.0000
C00653=-26.290,116.300,38.430,-0.0200,-0.0200,1.0000
C00654=-28.680,118.060,38.680,-0.0100,-0.0100,1.0000
C00655=-32.320,119.020,38.810,-0.0000,-0.0000,1.0000
C00656=-36.760,119.000,38.910,-0.0000,0.0100,1.0000
C00657=-41.300,117.920,39.020,0.0000,-0.0000,1.0000
C00658=-45.680,116.350,39.090,0.0000,-0.0000,1.0000
C00659=-49.970,114.570,39.090,0.0000,-0.0000,1.0000
C00660=-54.170,112.580,39.020,0.0000,-0.0000,1.0000
C00661=-58.150,110.140,38.910,-0.0100,0.0100,1.0000
C00662=-61.310,107.010,38.810,0.0000,-0.0000,1.0000
C00663=-63.200,103.760,38.680,0.0100,-0.0000,1.0000
C00664=-63.640,100.820,38.430,0.0300,-0.0000,1.0000
C00665=-63.510,97.970,37.930,0.0900,0.0100,1.0000
C00666=-63.480,95.260,37.260,0.2200,-0.0000,0.9800
C00667=-64.100,92.680,36.610,0.3800,-0.1200,0.9200
C00668=-66.050,89.880,36.120,0.4000,-0.3500,0.8400
C00669=-69.950,86.350,35.930,0.3700,-0.4300,0.8300
C00670=-74.230,82.670,35.920,0.3800,-0.4200,0.8300
C00671=-78.560,78.560,35.930,0.4000,-0.4000,0.8300
C00672=-82.670,74.230,35.920,0.4200,-0.3800,0.8300
C00673=-86.350,69.950,35.930,0.4300,-0.3700,0.8300
C00674=-89.880,66.050,36.120,0.3500,-0.4000,0.8400
C00675=-92.680,64.100,36.610,0.1200,-0.3800,0.9200
C00676=-95.260,63.480,37.260,0.0000,-0.2200,0.9800
C00677=-97.970,63.510,37.930,-0.0100,-0.0900,1.0000
C00678=-100.820,63.640,38.430,0.0000,-0.0300,1.0000
C00679=-103.760,63.200,38.680,0.0000,-0.0100,1.0000
C00680=-107.010,61.310,38.810,0.0000,-0.0000,1.0000
C00681=-110.140,58.150,38.910,-0.0100,0.0100,1.0000
C00682=-112.580,54.170,39.020,0.0000,-0.0000,1.0000
C00683=-114.570,49.970,39.090,0.0000,-0.0000,1.0000
C00684=-116.350,45.680,39.090,0.0000,-0.0000,1.0000
C00685=-117.920,41.300,39.020,0.0000,-0.0000,1.0000
C00686=-119.000,36.760,38.910,-0.0100,0.0000,1.0000
C00687=-119.020,32.320,38.810,0.0000,0.0000,1.0000
C00688=-118.060,28.680,38.680,0.0100,0.0100,1.0000
C00689=-116.300,26.290,38.430,0.0200,0.0200,1.0000
C00690=-114.180,24.360,37.930,0.0600,0.0700,1.0000
C00691=-112.250,22.470,37.260,0.1600,0.1500,0.9800
C00692=-110.860,20.210,36.610,0.3600,0.1800,0.9200
C00693=-110.260,16.850,36.120,0.5300,0.0400,0.8400
C00694=-110.520,11.600,35.930,0.5600,-0.0400,0.8300
C00695=-110.940,5.970,35.920,0.5600,-0.0300,0.8300
C00696=-111.100,0.000,35.930,0.5600,-0.0000,0.8300
C00697=-110.940,-5.970,35.920,0.5600,0.0300,0.8300
C00698=-110.520,-11.600,35.930,0.5600,0.0400,0.8300
C00699=-110.260,-16.850,36.120,0.5300,-0.0400,0.8400
C00700=-110.860,-20.210,36.610,0.3600,-0.1800,0.9200
C00701=-112.250,-22.470,37.260,0.1600,-0.1500,0.9800
C00702=-114.180,-24.360,37.930,0.0600,-0.0700,1.0000
C00703=-116.300,-26.290,38.430,0.0200,-0.0200,1.0000
C00704=-118.060,-28.680,38.680,0.0100,-0.0100,1.0000
C00705=-119.020,-32.320,38.810,0.0000,-0.0000,1.0000
C00706=-119.000,-36.760,38.910,-0.0100,-0.0000,1.0000
C00707=-117.920,-41.300,39.020,0.0000,0.0000,1.0000
C00708=-116.350,-45.680,39.090,0.0000,0.0000,1.0000
C00709=-114.570,-49.970,39.090,0.0000,0.0000,1.0000
C00710=-112.580,-54.170,39.020,0.0000,0.0000,1.0000
C00711=-110.140,-58.150,38.910,-0.0100,-0.0100,1.0000
C00712=-107.010,-61.310,38.810,0.0000,0.0000,1.0000
C00713=-103.760,-63.200,38.680,0.0000,0.0100,1.0000
C00714=-100.820,-63.640,38.430,0.0000,0.0300,1.0000
C00715=-97.970,-63.510,37.930,-0.0100,0.0900,1.0000
C00716=-95.260,-63.480,37.260,0.0000,0.2200,0.9800
C00717=-92.680,-64.100,36.610,0.1200,0.3800,0.9200
C00718=-89.880,-66.050,36.120,0.3500,0.4000,0.8400
C00719=-86.350,-69.950,35.930,0.4300,0.3700,0.8300
C00720=-82.670,-74.230,35.920,0.4200,0.3800,0.8300
C00721=-78.560,-78.560,35.930,0.4000,0.4000,0.8300
C00722=-74.230,-82.670,35.920,0.3800,0.4200,0.8300
C00723=-69.950,-86.350,35.930,0.3700,0.4300,0.8300
C00724=-66.050,-89.880,36.120,0.4000,0.3500,0.8400
C00725=-64.100,-92.680,36.610,0.3800,0.1200,0.9200
C00726=-63.480,-95.260,37.260,0.2200,0.0000,0.9800
C00727=-63.510,-97.970,37.930,0.0900,-0.0100,1.0000
C00728=-63.640,-100.820,38.430,0.0300,0.0000,1.0000
C00729=-63.200,-103.760,38.680,0.0100,0.0000,1.0000
C00730=-61.310,-107.010,38.810,0.0000,0.0000,1.0000
C00731=-58.150,-110.140,38.910,-0.0100,-0.0100,1.0000
C00732=-54.170,-112.580,39.020,0.0000,0.0000,1.0000
C00733=-49.970,-114.570,39.090,0.0000,0.0000,1.0000
C00734=-45.680,-116.350,39.090,0.0000,0.0000,1.0000
C00735=-41.300,-117.920,39.020,0.0000,0.0000,1.0000
C00736=-36.760,-119.000,38.910,-0.0000,-0.0100,1.0000
C00737=-32.320,-119.020,38.810,-0.0000,0.0000,1.0000
C00738=-28.680,-118.060,38.680,-0.0100,0.0100,1.0000
C00739=-26.290,-116.300,38.430,-0.0200,0.0200,1.0000
C00740=-24.360,-114.180,37.930,-0.0700,0.0600,1.0000
C00741=-22.470,-112.250,37.260,-0.1500,0.1600,0.9800
C00742=-20.210,-110.860,36.610,-0.1800,0.3600,0.9200
C00743=-16.850,-110.260,36.120,-0.0400,0.5300,0.8400
C00744=-11.600,-110.520,35.930,0.0400,0.5600,0.8300
C00745=-5.970,-110.940,35.920,0.0300,0.5600,0.8300
C00746=0.000,-111.100,35.930,0.0000,0.5600,0.8300
C00747=0.000,-111.100,35.930,0.0000,0.5600,0.8300
C00748=5.970,-110.940,35.920,-0.0300,0.5600,0.8300
C00749=11.600,-110.520,35.930,-0.0400,0.5600,0.8300
C00750=16.850,-110.260,36.120,0.0400,0.5300,0.8400
C00751=20.210,-110.860,36.610,0.1800,0.3600,0.9200
C00752=22.470,-112.250,37.260,0.1500,0.1600,0.9800
C00753=24.360,-114.180,37.930,0.0700,0.0600,1.0000
C00754=26.290,-116.300,38.430,0.0200,0.0200,1.0000
C00755=28.680,-118.060,38.680,0.0100,0.0100,1.0000
C00756=32.320,-119.020,38.810,0.0000,0.0000,1.0000
C00757=36.760,-119.000,38.910,0.0000,-0.0100,1.0000
C00758=41.300,-117.920,39.020,-0.0000,0.0000,1.0000
C00759=45.680,-116.350,39.090,-0.0000,0.0000,1.0000
C00760=49.970,-114.570,39.090,-0.0000,0.0000,1.0000
C00761=54.170,-112.580,39.020,-0.0000,0.0000,1.0000
C00762=58.150,-110.140,38.910,0.0100,-0.0100,1.0000
C00763=61.310,-107.010,38.810,-0.0000,0.0000,1.0000
C00764=63.200,-103.760,38.680,-0.0100,0.0000,1.0000
C00765=63.640,-100.820,38.430,-0.0300,0.0000,1.0000
C00766=63.510,-97.970,37.930,-0.0900,-0.0100,1.0000
C00767=63.480,-95.260,37.260,-0.2200,0.0000,0.9800
C00768=64.100,-92.680,36.610,-0.3800,0.1200,0.9200
C00769=66.050,-89.880,36.120,-0.4000,0.3500,0.8400
C00770=69.950,-86.350,35.930,-0.3700,0.4300,0.8300
C00771=74.230,-82.670,35.920,-0.3800,0.4200,0.8300
C00772=78.560,-78.560,35.930,-0.4000,0.4000,0.8300
C00773=82.670,-74.230,35.920,-0.4200,0.3800,0.8300
C00774=86.350,-69.950,35.930,-0.4300,0.3700,0.8300
C00775=89.880,-66.050,36.120,-0.3500,0.4000,0.8400
C00776=92.680,-64.100,36.610,-0.1200,0.3800,0.9200
C00777=95.260,-63.480,37.260,-0.0000,0.2200,0.9800
C00778=97.970,-63.510,37.930,0.0100,0.0900,1.0000
C00779=100.820,-63.640,38.430,-0.0000,0.0300,1.0000
C00780=103.760,-63.200,38.680,-0.0000,0.0100,1.0000
C00781=107.010,-61.310,38.810,-0.0000,0.0000,1.0000
C00782=110.140,-58.150,38.910,0.0100,-0.0100,1.0000
C00783=112.580,-54.170,39.020,-0.0000,0.0000,1.0000
C00784=114.570,-49.970,39.090,-0.0000,0.0000,1.0000
C00785=116.350,-45.680,39.090,-0.0000,0.0000,1.0000
C00786=117.920,-41.300,39.020,-0.0000,0.0000,1.0000
C00787=119.000,-36.760,38.910,0.0100,-0.0000,1.0000
C00788=119.020,-32.320,38.810,-0.0000,-0.0000,1.0000
C00789=118.060,-28.680,38.680,-0.0100,-0.0100,1.0000
C00790=116.300,-26.290,38.430,-0.0200,-0.0200,1.0000
C00791=114.180,-24.360,37.930,-0.0600,-0.0700,1.0000
C00792=112.250,-22.470,37.260,-0.1600,-0.1500,0.9800
C00793=110.860,-20.210,36.610,-0.3600,-0.1800,0.9200
C00794=110.260,-16.850,36.120,-0.5300,-0.0400,0.8400
C00795=110.520,-11.600,35.930,-0.5600,0.0400,0.8300
C00796=110.940,-5.970,35.920,-0.5600,0.0300,0.8300
C00797=111.100,0.000,35.930,-0.5600,0.0000,0.8300
C00798=110.940,5.970,35.920,-0.5600,-0.0300,0.8300
C00799=110.520,11.600,35.930,-0.5600,-0.0400,0.8300
C00800=110.260,16.850,36.120,-0.5300,0.0400,0.8400
C00801=110.860,20.210,36.610,-0.3600,0.1800,0.9200
C00802=112.250,22.470,37.260,-0.1600,0.1500,0.9800
C00803=114.180,24.360,37.930,-0.0600,0.0700,1.0000
C00804=116.300,26.290,38.430,-0.0200,0.0200,1.0000
C00805=118.060,28.680,38.680,-0.0100,0.0100,1.0000
C00806=119.020,32.320,38.810,-0.0000,0.0000,1.0000
C00807=119.000,36.760,38.910,0.0100,0.0000,1.0000
C00808=117.920,41.300,39.020,-0.0000,-0.0000,1.0000
C00809=116.350,45.680,39.090,-0.0000,-0.0000,1.0000
C00810=114.570,49.970,39.090,-0.0000,-0.0000,1.0000
C00811=112.580,54.170,39.020,-0.0000,-0.0000,1.0000
C00812=110.140,58.150,38.910,0.0100,0.0100,1.0000
C00813=107.010,61.310,38.810,-0.0000,-0.0000,1.0000
C00814=103.760,63.200,38.680,-0.0000,-0.0100,1.0000
C00815=100.820,63.640,38.430,-0.0000,-0.0300,1.0000
C00816=97.970,63.510,37.930,0.0100,-0.0900,1.0000
C00817=95.260,63.480,37.260,-0.0000,-0.2200,0.9800
C00818=92.680,64.100,36.610,-0.1200,-0.3800,0.9200
C00819=89.880,66.050,36.120,-0.3500,-0.4000,0.8400
C00820=86.350,69.950,35.930,-0.4300,-0.3700,0.8300
C00821=82.670,74.230,35.920,-0.4200,-0.3800,0.8300
C00822=78.560,78.560,35.930,-0.4000,-0.4000,0.8300
C00823=74.230,82.670,35.920,-0.3800,-0.4200,0.8300
C00824=69.950,86.350,35.930,-0.3700,-0.4300,0.8300
C00825=66.050,89.880,36.120,-0.4000,-0.3500,0.8400
C00826=64.100,92.680,36.610,-0.3800,-0.1200,0.9200
C00827=63.480,95.260,37.260,-0.2200,-0.0000,0.9800
C00828=63.510,97.970,37.930,-0.0900,0.0100,1.0000
C00829=63.640,100.820,38.430,-0.0300,-0.0000,1.0000
C00830=63.200,103.760,38.680,-0.0100,-0.0000,1.0000
C00831=61.310,107.010,38.810,-0.0000,-0.0000,1.0000
C00832=58.150,110.140,38.910,0.0100,0.0100,1.0000
C00833=54.170,112.580,39.020,-0.0000,-0.0000,1.0000
C00834=49.970,114.570,39.090,-0.0000,-0.0000,1.0000
C00835=45.680,116.350,39.090,-0.0000,-0.0000,1.0000
C00836=41.300,117.920,39.020,-0.0000,-0.0000,1.0000
C00837=36.760,119.000,38.910,0.0000,0.0100,1.0000
C00838=32.320,119.020,38.810,0.0000,-0.0000,1.0000
C00839=28.680,118.060,38.680,0.0100,-0.0100,1.0000
C00840=26.290,116.300,38.430,0.0200,-0.0200,1.0000
C00841=24.360,114.180,37.930,0.0700,-0.0600,1.0000
C00842=22.470,112.250,37.260,0.1500,-0.1600,0.9800
C00843=20.210,110.860,36.610,0.1800,-0.3600,0.9200
C00844=16.850,110.260,36.120,0.0400,-0.5300,0.8400
C00845=11.600,110.520,35.930,-0.0400,-0.5600,0.8300
C00846=5.970,110.940,35.920,-0.0300,-0.5600,0.8300
C00847=0.000,111.100,35.930,0.0000,-0.5600,0.8300
C00848=0.000,110.140,37.330,0.0000,-0.5700,0.8200
C00849=5.880,109.980,37.320,-0.0300,-0.5700,0.8200
C00850=11.450,109.560,37.330,-0.0400,-0.5700,0.8200
C00851=16.670,109.340,37.540,0.0500,-0.5400,0.8400
C00852=19.980,110.010,38.070,0.2000,-0.3400,0.9200
C00853=22.210,111.530,38.780,0.1500,-0.1400,0.9800
C00854=24.080,113.630,39.510,0.0600,-0.0400,1.0000
C00855=25.980,115.930,40.060,0.0100,-0.0100,1.0000
C00856=28.340,117.880,40.330,0.0000,-0.0000,1.0000
C00857=32.000,118.980,40.480,-0.0000,0.0000,1.0000
C00858=36.500,119.040,40.590,0.0000,0.0100,1.0000
C00859=41.140,117.970,40.710,-0.0000,-0.0000,1.0000
C00860=45.630,116.370,40.790,0.0000,0.0000,1.0000
C00861=50.020,114.550,40.790,0.0000,0.0000,1.0000
C00862=54.330,112.510,40.710,-0.0000,-0.0000,1.0000
C00863=58.370,109.990,40.590,0.0100,0.0100,1.0000
C00864=61.510,106.760,40.480,0.0000,0.0000,1.0000
C00865=63.310,103.390,40.330,-0.0000,-0.0000,1.0000
C00866=63.600,100.350,40.060,-0.0100,0.0000,1.0000
C00867=63.320,97.370,39.510,-0.0700,0.0100,1.0000
C00868=63.160,94.570,38.780,-0.2000,0.0100,0.9800
C00869=63.660,91.920,38.070,-0.3800,-0.1000,0.9200
C00870=65.530,89.100,37.540,-0.4100,-0.3500,0.8400
C00871=69.380,85.570,37.330,-0.3700,-0.4300,0.8200
C00872=73.610,81.930,37.320,-0.3800,-0.4300,0.8200
C00873=77.880,77.880,37.330,-0.4000,-0.4000,0.8200
C00874=81.930,73.610,37.320,-0.4300,-0.3800,0.8200
C00875=85.570,69.380,37.330,-0.4300,-0.3700,0.8200
C00876=89.100,65.530,37.540,-0.3500,-0.4100,0.8400
C00877=91.920,63.660,38.070,-0.1000,-0.3800,0.9200
C00878=94.570,63.160,38.780,0.0100,-0.2000,0.9800
C00879=97.370,63.320,39.510,0.0100,-0.0700,1.0000
C00880=100.350,63.600,40.060,0.0000,-0.0100,1.0000
C00881=103.390,63.310,40.330,-0.0000,-0.0000,1.0000
C00882=106.760,61.510,40.480,0.0000,0.0000,1.0000
C00883=109.990,58.370,40.590,0.0100,0.0100,1.0000
C00884=112.510,54.330,40.710,-0.0000,-0.0000,1.0000
C00885=114.550,50.020,40.790,0.0000,0.0000,1.0000
C00886=116.370,45.630,40.790,0.0000,0.0000,1.0000
C00887=117.970,41.140,40.710,-0.0000,-0.0000,1.0000
C00888=119.040,36.500,40.590,0.0100,0.0000,1.0000
C00889=118.980,32.000,40.480,0.0000,-0.0000,1.0000
C00890=117.880,28.340,40.330,-0.0000,0.0000,1.0000
C00891=115.930,25.980,40.060,-0.0100,0.0100,1.0000
C00892=113.630,24.080,39.510,-0.0400,0.0600,1.0000
C00893=111.530,22.210,38.780,-0.1400,0.1500,0.9800
C00894=110.010,19.980,38.070,-0.3400,0.2000,0.9200
C00895=109.340,16.670,37.540,-0.5400,0.0500,0.8400
C00896=109.560,11.450,37.330,-0.5700,-0.0400,0.8200
C00897=109.980,5.880,37.320,-0.5700,-0.0300,0.8200
C00898=110.140,0.000,37.330,-0.5700,0.0000,0.8200
C00899=109.980,-5.880,37.320,-0.5700,0.0300,0.8200
C00900=109.560,-11.450,37.330,-0.5700,0.0400,0.8200
C00901=109.340,-16.670,37.540,-0.5400,-0.0500,0.8400
C00902=110.010,-19.980,38.070,-0.3400,-0.2000,0.9200
C00903=111.530,-22.210,38.780,-0.1400,-0.1500,0.9800
C00904=113.630,-24.080,39.510,-0.0400,-0.0600,1.0000
C00905=115.930,-25.980,40.060,-0.0100,-0.0100,1.0000
C00906=117.880,-28.340,40.330,-0.0000,-0.0000,1.0000
C00907=118.980,-32.000,40.480,0.0000,0.0000,1.0000
C00908=119.040,-36.500,40.590,0.0100,-0.0000,1.0000
C00909=117.970,-41.140,40.710,-0.0000,0.0000,1.0000
C00910=116.370,-45.630,40.790,0.0000,-0.0000,1.0000
C00911=114.550,-50.020,40.790,0.0000,-0.0000,1.0000
C00912=112.510,-54.330,40.710,-0.0000,0.0000,1.0000
C00913=109.990,-58.370,40.590,0.0100,-0.0100,1.0000
C00914=106.760,-61.510,40.480,0.0000,-0.0000,1.0000
C00915=103.390,-63.310,40.330,-0.0000,0.0000,1.0000
C00916=100.350,-63.600,40.060,0.0000,0.0100,1.0000
C00917=97.370,-63.320,39.510,0.0100,0.0700,1.0000
C00918=94.570,-63.160,38.780,0.0100,0.2000,0.9800
C00919=91.920,-63.660,38.070,-0.1000,0.3800,0.9200
C00920=89.100,-65.530,37.540,-0.3500,0.4100,0.8400
C00921=85.570,-69.380,37.330,-0.4300,0.3700,0.8200
C00922=81.930,-73.610,37.320,-0.4300,0.3800,0.8200
C00923=77.880,-77.880,37.330,-0.4000,0.4000,0.8200
C00924=73.610,-81.930,37.320,-0.3800,0.4300,0.8200
C00925=69.380,-85.570,37.330,-0.3700,0.4300,0.8200
C00926=65.530,-89.100,37.540,-0.4100,0.3500,0.8400
C00927=63.660,-91.920,38.070,-0.3800,0.1000,0.9200
C00928=63.160,-94.570,38.780,-0.2000,-0.0100,0.9800
C00929=63.320,-97.370,39.510,-0.0700,-0.0100,1.0000
C00930=63.600,-100.350,40.060,-0.0100,-0.0000,1.0000
C00931=63.310,-103.390,40.330,-0.0000,0.0000,1.0000
C00932=61.510,-106.760,40.480,0.0000,-0.0000,1.0000
C00933=58.370,-109.990,40.590,0.0100,-0.0100,1.0000
C00934=54.330,-112.510,40.710,-0.0000,0.0000,1.0000
C00935=50.020,-114.550,40.790,0.0000,-0.0000,1.0000
C00936=45.630,-116.370,40.790,0.0000,-0.0000,1.0000
C00937=41.140,-117.970,40.710,-0.0000,0.0000,1.0000
C00938=36.500,-119.040,40.590,0.0000,-0.0100,1.0000
C00939=32.000,-118.980,40.480,-0.0000,-0.0000,1.0000
C00940=28.340,-117.880,40.330,0.0000,0.0000,1.0000
C00941=25.980,-115.930,40.060,0.0100,0.0100,1.0000
C00942=24.080,-113.630,39.510,0.0600,0.0400,1.0000
C00943=22.210,-111.530,38.780,0.1500,0.1400,0.9800
C00944=19.980,-110.010,38.070,0.2000,0.3400,0.9200
C00945=16.670,-109.340,37.540,0.0500,0.5400,0.8400
C00946=11.450,-109.560,37.330,-0.0400,0.5700,0.8200
C00947=5.880,-109.980,37.320,-0.0300,0.5700,0.8200
C00948=0.000,-110.140,37.330,0.0000,0.5700,0.8200
C00949=0.000,-110.140,37.330,0.0000,0.5700,0.8200
C00950=-5.880,-109.980,37.320,0.0300,0.5700,0.8200
C00951=-11.450,-109.560,37.330,0.0400,0.5700,0.8200
C00952=-16.670,-109.340,37.540,-0.0500,0.5400,0.8400
C00953=-19.980,-110.010,38.070,-0.2000,0.3400,0.9200
C00954=-22.210,-111.530,38.780,-0.1500,0.1400,0.9800
C00955=-24.080,-113.630,39.510,-0.0600,0.0400,1.0000
C00956=-25.980,-115.930,40.060,-0.0100,0.0100,1.0000
C00957=-28.340,-117.880,40.330,-0.0000,0.0000,1.0000
C00958=-32.000,-118.980,40.480,0.0000,-0.0000,1.0000
C00959=-36.500,-119.040,40.590,-0.0000,-0.0100,1.0000
C00960=-41.140,-117.970,40.710,0.0000,0.0000,1.0000
C00961=-45.630,-116.370,40.790,-0.0000,-0.0000,1.0000
C00962=-50.020,-114.550,40.790,-0.0000,-0.0000,1.0000
C00963=-54.330,-112.510,40.710,0.0000,0.0000,1.0000
C00964=-58.370,-109.990,40.590,-0.0100,-0.0100,1.0000
C00965=-61.510,-106.760,40.480,-0.0000,-0.0000,1.0000
C00966=-63.310,-103.390,40.330,0.0000,0.0000,1.0000
C00967=-63.600,-100.350,40.060,0.0100,-0.0000,1.0000
C00968=-63.320,-97.370,39.510,0.0700,-0.0100,1.0000
C00969=-63.160,-94.570,38.780,0.2000,-0.0100,0.9800
C00970=-63.660,-91.920,38.070,0.3800,0.1000,0.9200
C00971=-65.530,-89.100,37.540,0.4100,0.3500,0.8400
C00972=-69.380,-85.570,37.330,0.3700,0.4300,0.8200
C00973=-73.610,-81.930,37.320,0.3800,0.4300,0.8200
C00974=-77.880,-77.880,37.330,0.4000,0.4000,0.8200
C00975=-81.930,-73.610,37.320,0.4300,0.3800,0.8200
C00976=-85.570,-69.380,37.330,0.4300,0.3700,0.8200
C00977=-89.100,-65.530,37.540,0.3500,0.4100,0.8400
C00978=-91.920,-63.660,38.070,0.1000,0.3800,0.9200
C00979=-94.570,-63.160,38.780,-0.0100,0.2000,0.9800
C00980=-97.370,-63.320,39.510,-0.0100,0.0700,1.0000
C00981=-100.350,-63.600,40.060,-0.0000,0.0100,1.0000
C00982=-103.390,-63.310,40.330,0.0000,0.0000,1.0000
C00983=-106.760,-61.510,40.480,-0.0000,-0.0000,1.0000
C00984=-109.990,-58.370,40.590,-0.0100,-0.0100,1.0000
C00985=-112.510,-54.330,40.710,0.0000,0.0000,1.0000
C00986=-114.550,-50.020,40.790,-0.0000,-0.0000,1.0000
C00987=-116.370,-45.630,40.790,-0.0000,-0.0000,1.0000
C00988=-117.970,-41.140,40.710,0.0000,0.0000,1.0000
C00989=-119.040,-36.500,40.590,-0.0100,-0.0000,1.0000
C00990=-118.980,-32.000,40.480,-0.0000,0.0000,1.0000
C00991=-117.880,-28.340,40.330,0.0000,-0.0000,1.0000
C00992=-115.930,-25.980,40.060,0.0100,-0.0100,1.0000
C00993=-113.630,-24.080,39.510,0.0400,-0.0600,1.0000
C00994=-111.530,-22.210,38.780,0.1400,-0.1500,0.9800
C00995=-110.010,-19.980,38.070,0.3400,-0.2000,0.9200
C00996=-109.340,-16.670,37.540,0.5400,-0.0500,0.8400
C00997=-109.560,-11.450,37.330,0.5700,0.0400,0.8200
C00998=-109.980,-5.880,37.320,0.5700,0.0300,0.8200
C00999=-110.140,0.000,37.330,0.5700,-0.0000,0.8200
C01000=-109.980,5.880,37.320,0.5700,-0.0300,0.8200
C01001=-109.560,11.450,37.330,0.5700,-0.0400,0.8200
C01002=-109.340,16.670,37.540,0.5400,0.0500,0.8400
C01003=-110.010,19.980,38.070,0.3400,0.2000,0.9200
C01004=-111.530,22.210,38.780,0.1400,0.1500,0.9800
C01005=-113.630,24.080,39.510,0.0400,0.0600,1.0000
C01006=-115.930,25.980,40.060,0.0100,0.0100,1.0000
C01007=-117.880,28.340,40.330,0.0000,0.0000,1.0000
C01008=-118.980,32.000,40.480,-0.0000,-0.0000,1.0000
C01009=-119.040,36.500,40.590,-0.0100,0.0000,1.0000
C01010=-117.970,41.140,40.710,0.0000,-0.0000,1.0000
C01011=-116.370,45.630,40.790,-0.0000,0.0000,1.0000
C01012=-114.550,50.020,40.790,-0.0000,0.0000,1.0000
C01013=-112.510,54.330,40.710,0.0000,-0.0000,1.0000
C01014=-109.990,58.370,40.590,-0.0100,0.0100,1.0000
C01015=-106.760,61.510,40.480,-0.0000,0.0000,1.0000
C01016=-103.390,63.310,40.330,0.0000,-0.0000,1.0000
C01017=-100.350,63.600,40.060,-0.0000,-0.0100,1.0000
C01018=-97.370,63.320,39.510,-0.0100,-0.0700,1.0000
C01019=-94.570,63.160,38.780,-0.0100,-0.2000,0.9800
C01020=-91.920,63.660,38.070,0.1000,-0.3800,0.9200
C01021=-89.100,65.530,37.540,0.3500,-0.4100,0.8400
C01022=-85.570,69.380,37.330,0.4300,-0.3700,0.8200
C01023=-81.930,73.610,37.320,0.4300,-0.3800,0.8200
C01024=-77.880,77.880,37.330,0.4000,-0.4000,0.8200
C01025=-73.610,81.930,37.320,0.3800,-0.4300,0.8200
C01026=-69.380,85.570,37.330,0.3700,-0.4300,0.8200
C01027=-65.530,89.100,37.540,0.4100,-0.3500,0.8400
C01028=-63.660,91.920,38.070,0.3800,-0.1000,0.9200
C01029=-63.160,94.570,38.780,0.2000,0.0100,0.9800
C01030=-63.320,97.370,39.510,0.0700,0.0100,1.0000
C01031=-63.600,100.350,40.060,0.0100,0.0000,1.0000
C01032=-63.310,103.390,40.330,0.0000,-0.0000,1.0000
C01033=-61.510,106.760,40.480,-0.0000,0.0000,1.0000
C01034=-58.370,109.990,40.590,-0.0100,0.0100,1.0000
C01035=-54.330,112.510,40.710,0.0000,-0.0000,1.0000
C01036=-50.020,114.550,40.790,-0.0000,0.0000,1.0000
C01037=-45.630,116.370,40.790,-0.0000,0.0000,1.0000
C01038=-41.140,117.970,40.710,0.0000,-0.0000,1.0000
C01039=-36.500,119.040,40.590,-0.0000,0.0100,1.0000
C01040=-32.000,118.980,40.480,0.0000,0.0000,1.0000
C01041=-28.340,117.880,40.330,-0.0000,-0.0000,1.0000
C01042=-25.980,115.930,40.060,-0.0100,-0.0100,1.0000
C01043=-24.080,113.630,39.510,-0.0600,-0.0400,1.0000
C01044=-22.210,111.530,38.780,-0.1500,-0.1400,0.9800
C01045=-19.980,110.010,38.070,-0.2000,-0.3400,0.9200
C01046=-16.670,109.340,37.540,-0.0500,-0.5400,0.8400
C01047=-11.450,109.560,37.330,0.0400,-0.5700,0.8200
C01048=-5.880,109.980,37.320,0.0300,-0.5700,0.8200
C01049=0.000,110.140,37.330,0.0000,-0.5700,0.8200
C01050=0.000,109.160,38.720,0.0000,-0.5800,0.8100
C01051=-5.790,109.000,38.710,0.0300,-0.5800,0.8100
C01052=-11.300,108.600,38.720,0.0400,-0.5800,0.8200
C01053=-16.480,108.400,38.950,-0.0600,-0.5500,0.8400
C01054=-19.750,109.160,39.520,-0.2100,-0.3300,0.9200
C01055=-21.950,110.800,40.290,-0.1400,-0.1200,0.9800
C01056=-23.790,113.060,41.090,-0.0500,-0.0300,1.0000
C01057=-25.670,115.560,41.690,0.0000,0.0000,1.0000
C01058=-28.000,117.690,41.990,0.0000,0.0100,1.0000
C01059=-31.670,118.950,42.150,0.0000,0.0100,1.0000
C01060=-36.250,119.090,42.270,-0.0000,0.0100,1.0000
C01061=-40.980,118.020,42.400,-0.0000,0.0000,1.0000
C01062=-45.570,116.390,42.490,-0.0000,0.0000,1.0000
C01063=-50.080,114.520,42.490,-0.0000,0.0000,1.0000
C01064=-54.480,112.430,42.400,-0.0000,0.0000,1.0000
C01065=-58.580,109.840,42.270,-0.0100,0.0100,1.0000
C01066=-61.710,106.500,42.150,-0.0100,0.0100,1.0000
C01067=-63.420,103.020,41.990,-0.0100,0.0000,1.0000
C01068=-63.560,99.860,41.690,-0.0000,-0.0000,1.0000
C01069=-63.130,96.770,41.090,0.0600,0.0100,1.0000
C01070=-62.820,93.860,40.290,0.1800,0.0100,0.9800
C01071=-63.220,91.150,39.520,0.3800,-0.0800,0.9200
C01072=-65.000,88.310,38.950,0.4300,-0.3500,0.8400
C01073=-68.800,84.780,38.720,0.3800,-0.4400,0.8200
C01074=-72.980,81.170,38.710,0.3900,-0.4300,0.8100
C01075=-77.190,77.190,38.720,0.4100,-0.4100,0.8100
C01076=-81.170,72.980,38.710,0.4300,-0.3900,0.8100
C01077=-84.780,68.800,38.720,0.4400,-0.3800,0.8200
C01078=-88.310,65.000,38.950,0.3500,-0.4300,0.8400
C01079=-91.150,63.220,39.520,0.0800,-0.3800,0.9200
C01080=-93.860,62.820,40.290,-0.0100,-0.1800,0.9800
C01081=-96.770,63.130,41.090,-0.0100,-0.0600,1.0000
C01082=-99.860,63.560,41.690,0.0000,0.0000,1.0000
C01083=-103.020,63.420,41.990,-0.0000,0.0100,1.0000
C01084=-106.500,61.710,42.150,-0.0100,0.0100,1.0000
C01085=-109.840,58.580,42.270,-0.0100,0.0100,1.0000
C01086=-112.430,54.480,42.400,-0.0000,0.0000,1.0000
C01087=-114.520,50.080,42.490,-0.0000,0.0000,1.0000
C01088=-116.390,45.570,42.490,-0.0000,0.0000,1.0000
C01089=-118.020,40.980,42.400,-0.0000,0.0000,1.0000
C01090=-119.090,36.250,42.270,-0.0100,0.0000,1.0000
C01091=-118.950,31.670,42.150,-0.0100,-0.0000,1.0000
C01092=-117.690,28.000,41.990,-0.0100,-0.0000,1.0000
C01093=-115.560,25.670,41.690,-0.0000,-0.0000,1.0000
C01094=-113.060,23.790,41.090,0.0300,0.0500,1.0000
C01095=-110.800,21.950,40.290,0.1200,0.1400,0.9800
C01096=-109.160,19.750,39.520,0.3300,0.2100,0.9200
C01097=-108.400,16.480,38.950,0.5500,0.0600,0.8400
C01098=-108.600,11.300,38.720,0.5800,-0.0400,0.8200
C01099=-109.000,5.790,38.710,0.5800,-0.0300,0.8100
C01100=-109.160,0.000,38.720,0.5800,-0.0000,0.8100
C01101=-109.000,-5.790,38.710,0.5800,0.0300,0.8100
C01102=-108.600,-11.300,38.720,0.5800,0.0400,0.8200
C01103=-108.400,-16.480,38.950,0.5500,-0.0600,0.8400
C01104=-109.160,-19.750,39.520,0.3300,-0.2100,0.9200
C01105=-110.800,-21.950,40.290,0.1200,-0.1400,0.9800
C01106=-113.060,-23.790,41.090,0.0300,-0.0500,1.0000
C01107=-115.560,-25.670,41.690,-0.0000,0.0000,1.0000
C01108=-117.690,-28.000,41.990,-0.0100,0.0000,1.0000
C01109=-118.950,-31.670,42.150,-0.0100,0.0000,1.0000
C01110=-119.090,-36.250,42.270,-0.0100,-0.0000,1.0000
C01111=-118.020,-40.980,42.400,-0.0000,-0.0000,1.0000
C01112=-116.390,-45.570,42.490,-0.0000,-0.0000,1.0000
C01113=-114.520,-50.080,42.490,-0.0000,-0.0000,1.0000
C01114=-112.430,-54.480,42.400,-0.0000,-0.0000,1.0000
C01115=-109.840,-58.580,42.270,-0.0100,-0.0100,1.0000
C01116=-106.500,-61.710,42.150,-0.0100,-0.0100,1.0000
C01117=-103.020,-63.420,41.990,-0.0000,-0.0100,1.0000
C01118=-99.860,-63.560,41.690,0.0000,-0.0000,1.0000
C01119=-96.770,-63.130,41.090,-0.0100,0.0600,1.0000
C01120=-93.860,-62.820,40.290,-0.0100,0.1800,0.9800
C01121=-91.150,-63.220,39.520,0.0800,0.3800,0.9200
C01122=-88.310,-65.000,38.950,0.3500,0.4300,0.8400
C01123=-84.780,-68.800,38.720,0.4400,0.3800,0.8200
C01124=-81.170,-72.980,38.710,0.4300,0.3900,0.8100
C01125=-77.190,-77.190,38.720,0.4100,0.4100,0.8100
C01126=-72.980,-81.170,38.710,0.3900,0.4300,0.8100
C01127=-68.800,-84.780,38.720,0.3800,0.4400,0.8200
C01128=-65.000,-88.310,38.950,0.4300,0.3500,0.8400
C01129=-63.220,-91.150,39.520,0.3800,0.0800,0.9200
C01130=-62.820,-93.860,40.290,0.1800,-0.0100,0.9800
C01131=-63.130,-96.770,41.090,0.0600,-0.0100,1.0000
C01132=-63.560,-99.860,41.690,-0.0000,0.0000,1.0000
C01133=-63.420,-103.020,41.990,-0.0100,-0.0000,1.0000
C01134=-61.710,-106.500,42.150,-0.0100,-0.0100,1.0000
C01135=-58.580,-109.840,42.270,-0.0100,-0.0100,1.0000
C01136=-54.480,-112.430,42.400,-0.0000,-0.0000,1.0000
C01137=-50.080,-114.520,42.490,-0.0000,-0.0000,1.0000
C01138=-45.570,-116.390,42.490,-0.0000,-0.0000,1.0000
C01139=-40.980,-118.020,42.400,-0.0000,-0.0000,1.0000
C01140=-36.250,-119.090,42.270,-0.0000,-0.0100,1.0000
C01141=-31.670,-118.950,42.150,0.0000,-0.0100,1.0000
C01142=-28.000,-117.690,41.990,0.0000,-0.0100,1.0000
C01143=-25.670,-115.560,41.690,0.0000,-0.0000,1.0000
C01144=-23.790,-113.060,41.090,-0.0500,0.0300,1.0000
C01145=-21.950,-110.800,40.290,-0.1400,0.1200,0.9800
C01146=-19.750,-109.160,39.520,-0.2100,0.3300,0.9200
C01147=-16.480,-108.400,38.950,-0.0600,0.5500,0.8400
C01148=-11.300,-108.600,38.720,0.0400,0.5800,0.8200
C01149=-5.790,-109.000,38.710,0.0300,0.5800,0.8100
C01150=0.000,-109.160,38.720,0.0000,0.5800,0.8100
C01151=0.000,-109.160,38.720,0.0000,0.5800,0.8100
C01152=5.790,-109.000,38.710,-0.0300,0.5800,0.8100
C01153=11.300,-108.600,38.720,-0.0400,0.5800,0.8200
C01154=16.480,-108.400,38.950,0.0600,0.5500,0.8400
C01155=19.750,-109.160,39.520,0.2100,0.3300,0.9200
C01156=21.950,-110.800,40.290,0.1400,0.1200,0.9800
C01157=23.790,-113.060,41.090,0.0500,0.0300,1.0000
C01158=25.670,-115.560,41.690,-0.0000,-0.0000,1.0000
C01159=28.000,-117.690,41.990,-0.0000,-0.0100,1.0000
C01160=31.670,-118.950,42.150,-0.0000,-0.0100,1.0000
C01161=36.250,-119.090,42.270,0.0000,-0.0100,1.0000
C01162=40.980,-118.020,42.400,0.0000,-0.0000,1.0000
C01163=45.570,-116.390,42.490,0.0000,-0.0000,1.0000
C01164=50.080,-114.520,42.490,0.0000,-0.0000,1.0000
C01165=54.480,-112.430,42.400,0.0000,-0.0000,1.0000
C01166=58.580,-109.840,42.270,0.0100,-0.0100,1.0000
C01167=61.710,-106.500,42.150,0.0100,-0.0100,1.0000
C01168=63.420,-103.020,41.990,0.0100,-0.0000,1.0000
C01169=63.560,-99.860,41.690,0.0000,0.0000,1.0000
C01170=63.130,-96.770,41.090,-0.0600,-0.0100,1.0000
C01171=62.820,-93.860,40.290,-0.1800,-0.0100,0.9800
C01172=63.220,-91.150,39.520,-0.3800,0.0800,0.9200
C01173=65.000,-88.310,38.950,-0.4300,0.3500,0.8400
C01174=68.800,-84.780,38.720,-0.3800,0.4400,0.8200
C01175=72.980,-81.170,38.710,-0.3900,0.4300,0.8100
C01176=77.190,-77.190,38.720,-0.4100,0.4100,0.8100
C01177=81.170,-72.980,38.710,-0.4300,0.3900,0.8100
C01178=84.780,-68.800,38.720,-0.4400,0.3800,0.8200
C01179=88.310,-65.000,38.950,-0.3500,0.4300,0.8400
C01180=91.150,-63.220,39.520,-0.0800,0.3800,0.9200
C01181=93.860,-62.820,40.290,0.0100,0.1800,0.9800
C01182=96.770,-63.130,41.090,0.0100,0.0600,1.0000
C01183=99.860,-63.560,41.690,-0.0000,-0.0000,1.0000
C01184=103.020,-63.420,41.990,0.0000,-0.0100,1.0000
C01185=106.500,-61.710,42.150,0.0100,-0.0100,1.0000
C01186=109.840,-58.580,42.270,0.0100,-0.0100,1.0000
C01187=112.430,-54.480,42.400,0.0000,-0.0000,1.0000
C01188=114.520,-50.080,42.490,0.0000,-0.0000,1.0000
C01189=116.390,-45.570,42.490,0.0000,-0.0000,1.0000
C01190=118.020,-40.980,42.400,0.0000,-0.0000,1.0000
C01191=119.090,-36.250,42.270,0.0100,-0.0000,1.0000
C01192=118.950,-31.670,42.150,0.0100,0.0000,1.0000
C01193=117.690,-28.000,41.990,0.0100,0.0000,1.0000
C01194=115.560,-25.670,41.690,0.0000,0.0000,1.0000
C01195=113.060,-23.790,41.090,-0.0300,-0.0500,1.0000
C01196=110.800,-21.950,40.290,-0.1200,-0.1400,0.9800
C01197=109.160,-19.750,39.520,-0.3300,-0.2100,0.9200
C01198=108.400,-16.480,38.950,-0.5500,-0.0600,0.8400
C01199=108.600,-11.300,38.720,-0.5800,0.0400,0.8200
C01200=109.000,-5.790,38.710,-0.5800,0.0300,0.8100
C01201=109.160,0.000,38.720,-0.5800,0.0000,0.8100
C01202=109.000,5.790,38.710,-0.5800,-0.0300,0.8100
C01203=108.600,11.300,38.720,-0.5800,-0.0400,0.8200
C01204=108.400,16.480,38.950,-0.5500,0.0600,0.8400
C01205=109.160,19.750,39.520,-0.3300,0.2100,0.9200
C01206=110.800,21.950,40.290,-0.1200,0.1400,0.9800
C01207=113.060,23.790,41.090,-0.0300,0.0500,1.0000
C01208=115.560,25.670,41.690,0.0000,-0.0000,1.0000
C01209=117.690,28.000,41.990,0.0100,-0.0000,1.0000
C01210=118.950,31.670,42.150,0.0100,-0.0000,1.0000
C01211=119.090,36.250,42.270,0.0100,0.0000,1.0000
C01212=118.020,40.980,42.400,0.0000,0.0000,1.0000
C01213=116.390,45.570,42.490,0.0000,0.0000,1.0000
C01214=114.520,50.080,42.490,0.0000,0.0000,1.0000
C01215=112.430,54.480,42.400,0.0000,0.0000,1.0000
C01216=109.840,58.580,42.270,0.0100,0.0100,1.0000
C01217=106.500,61.710,42.150,0.0100,0.0100,1.0000
C01218=103.020,63.420,41.990,0.0000,0.0100,1.0000
C01219=99.860,63.560,41.690,-0.0000,0.0000,1.0000
C01220=96.770,63.130,41.090,0.0100,-0.0600,1.0000
C01221=93.860,62.820,40.290,0.0100,-0.1800,0.9800
C01222=91.150,63.220,39.520,-0.0800,-0.3800,0.9200
C01223=88.310,65.000,38.950,-0.3500,-0.4300,0.8400
C01224=84.780,68.800,38.720,-0.4400,-0.3800,0.8200
C01225=81.170,72.980,38.710,-0.4300,-0.3900,0.8100
C01226=77.190,77.190,38.720,-0.4100,-0.4100,0.8100
C01227=72.980,81.170,38.710,-0.3900,-0.4300,0.8100
C01228=68.800,84.780,38.720,-0.3800,-0.4400,0.8200
C01229=65.000,88.310,38.950,-0.4300,-0.3500,0.8400
C01230=63.220,91.150,39.520,-0.3800,-0.0800,0.9200
C01231=62.820,93.860,40.290,-0.1800,0.0100,0.9800
C01232=63.130,96.770,41.090,-0.0600,0.0100,1.0000
C01233=63.560,99.860,41.690,0.0000,-0.0000,1.0000
C01234=63.420,103.020,41.990,0.0100,0.0000,1.0000
C01235=61.710,106.500,42.150,0.0100,0.0100,1.0000
C01236=58.580,109.840,42.270,0.0100,0.0100,1.0000
C01237=54.480,112.430,42.400,0.0000,0.0000,1.0000
C01238=50.080,114.520,42.490,0.0000,0.0000,1.0000
C01239=45.570,116.390,42.490,0.0000,0.0000,1.0000
C01240=40.980,118.020,42.400,0.0000,0.0000,1.0000
C01241=36.250,119.090,42.270,0.0000,0.0100,1.0000
C01242=31.670,118.950,42.150,-0.0000,0.0100,1.0000
C01243=28.000,117.690,41.990,-0.0000,0.0100,1.0000
C01244=25.670,115.560,41.690,-0.0000,0.0000,1.0000
C01245=23.790,113.060,41.090,0.0500,-0.0300,1.0000
C01246=21.950,110.800,40.290,0.1400,-0.1200,0.9800
C01247=19.750,109.160,39.520,0.2100,-0.3300,0.9200
C01248=16.480,108.400,38.950,0.0600,-0.5500,0.8400
C01249=11.300,108.600,38.720,-0.0400,-0.5800,0.8200
C01250=5.790,109.000,38.710,-0.0300,-0.5800,0.8100
C01251=0.000,109.160,38.720,0.0000,-0.5800,0.8100
C01252=0.000,108.170,40.100,0.0000,-0.5900,0.8100
C01253=5.700,108.010,40.090,-0.0300,-0.5900,0.8100
C01254=11.150,107.620,40.100,-0.0400,-0.5800,0.8100
C01255=16.290,107.460,40.350,0.0700,-0.5500,0.8300
C01256=19.520,108.290,40.960,0.2200,-0.3100,0.9300
C01257=21.680,110.050,41.800,0.1300,-0.1100,0.9900
C01258=23.490,112.490,42.660,0.0400,-0.0200,1.0000
C01259=25.350,115.170,43.320,-0.0100,0.0100,1.0000
C01260=27.650,117.500,43.640,-0.0100,0.0200,1.0000
C01261=31.340,118.910,43.810,-0.0000,0.0100,1.0000
C01262=35.980,119.140,43.950,0.0000,0.0200,1.0000
C01263=40.810,118.080,44.090,0.0000,0.0000,1.0000
C01264=45.510,116.410,44.190,0.0000,0.0000,1.0000
C01265=50.130,114.500,44.190,0.0000,0.0000,1.0000
C01266=54.640,112.350,44.090,0.0000,0.0000,1.0000
C01267=58.800,109.690,43.950,0.0100,0.0100,1.0000
C01268=61.920,106.240,43.810,0.0100,0.0100,1.0000
C01269=63.530,102.640,43.640,0.0200,0.0000,1.0000
C01270=63.520,99.360,43.320,0.0100,-0.0000,1.0000
C01271=62.930,96.150,42.660,-0.0400,0.0100,1.0000
C01272=62.490,93.150,41.800,-0.1700,0.0200,0.9900
C01273=62.770,90.380,40.960,-0.3700,-0.0700,0.9300
C01274=64.460,87.500,40.350,-0.4300,-0.3400,0.8300
C01275=68.210,83.980,40.100,-0.3900,-0.4400,0.8100
C01276=72.340,80.410,40.090,-0.3900,-0.4400,0.8100
C01277=76.490,76.490,40.100,-0.4200,-0.4200,0.8100
C01278=80.410,72.350,40.090,-0.4400,-0.3900,0.8100
C01279=83.980,68.210,40.100,-0.4400,-0.3900,0.8100
C01280=87.500,64.460,40.350,-0.3400,-0.4300,0.8300
C01281=90.380,62.770,40.960,-0.0700,-0.3700,0.9300
C01282=93.150,62.490,41.800,0.0200,-0.1700,0.9900
C01283=96.150,62.930,42.660,0.0100,-0.0400,1.0000
C01284=99.360,63.520,43.320,-0.0000,0.0100,1.0000
C01285=102.640,63.530,43.640,0.0000,0.0200,1.0000
C01286=106.240,61.920,43.810,0.0100,0.0100,1.0000
C01287=109.690,58.800,43.950,0.0100,0.0100,1.0000
C01288=112.350,54.640,44.090,0.0000,0.0000,1.0000
C01289=114.500,50.130,44.190,0.0000,0.0000,1.0000
C01290=116.410,45.510,44.190,0.0000,0.0000,1.0000
C01291=118.080,40.810,44.090,0.0000,0.0000,1.0000
C01292=119.140,35.980,43.950,0.0200,0.0000,1.0000
C01293=118.910,31.340,43.810,0.0100,-0.0000,1.0000
C01294=117.500,27.650,43.640,0.0200,-0.0100,1.0000
C01295=115.170,25.350,43.320,0.0100,-0.0100,1.0000
C01296=112.490,23.490,42.660,-0.0200,0.0400,1.0000
C01297=110.050,21.680,41.800,-0.1100,0.1300,0.9900
C01298=108.290,19.520,40.960,-0.3100,0.2200,0.9300
C01299=107.460,16.290,40.350,-0.5500,0.0700,0.8300
C01300=107.620,11.150,40.100,-0.5800,-0.0400,0.8100
C01301=108.010,5.700,40.090,-0.5900,-0.0300,0.8100
C01302=108.170,0.000,40.100,-0.5900,0.0000,0.8100
C01303=108.010,-5.700,40.090,-0.5900,0.0300,0.8100
C01304=107.620,-11.150,40.100,-0.5800,0.0400,0.8100
C01305=107.460,-16.290,40.350,-0.5500,-0.0700,0.8300
C01306=108.290,-19.520,40.960,-0.3100,-0.2200,0.9300
C01307=110.050,-21.680,41.800,-0.1100,-0.1300,0.9900
C01308=112.490,-23.490,42.660,-0.0200,-0.0400,1.0000
C01309=115.170,-25.350,43.320,0.0100,0.0100,1.0000
C01310=117.500,-27.650,43.640,0.0200,0.0100,1.0000
C01311=118.910,-31.340,43.810,0.0100,0.0000,1.0000
C01312=119.140,-35.980,43.950,0.0200,-0.0000,1.0000
C01313=118.080,-40.810,44.090,0.0000,-0.0000,1.0000
C01314=116.410,-45.510,44.190,0.0000,-0.0000,1.0000
C01315=114.500,-50.130,44.190,0.0000,-0.0000,1.0000
C01316=112.350,-54.640,44.090,0.0000,-0.0000,1.0000
C01317=109.690,-58.800,43.950,0.0100,-0.0100,1.0000
C01318=106.240,-61.920,43.810,0.0100,-0.0100,1.0000
C01319=102.640,-63.530,43.640,0.0000,-0.0200,1.0000
C01320=99.360,-63.520,43.320,-0.0000,-0.0100,1.0000
C01321=96.150,-62.930,42.660,0.0100,0.0400,1.0000
C01322=93.150,-62.490,41.800,0.0200,0.1700,0.9900
C01323=90.380,-62.770,40.960,-0.0700,0.3700,0.9300
C01324=87.500,-64.460,40.350,-0.3400,0.4300,0.8300
C01325=83.980,-68.210,40.100,-0.4400,0.3900,0.8100
C01326=80.410,-72.340,40.090,-0.4400,0.3900,0.8100
C01327=76.490,-76.490,40.100,-0.4200,0.4200,0.8100
C01328=72.350,-80.410,40.090,-0.3900,0.4400,0.8100
C01329=68.210,-83.980,40.100,-0.3900,0.4400,0.8100
C01330=64.460,-87.500,40.350,-0.4300,0.3400,0.8300
C01331=62.770,-90.380,40.960,-0.3700,0.0700,0.9300
C01332=62.490,-93.150,41.800,-0.1700,-0.0200,0.9900
C01333=62.930,-96.150,42.660,-0.0400,-0.0100,1.0000
C01334=63.520,-99.360,43.320,0.0100,0.0000,1.0000
C01335=63.530,-102.640,43.640,0.0200,-0.0000,1.0000
C01336=61.920,-106.240,43.810,0.0100,-0.0100,1.0000
C01337=58.800,-109.690,43.950,0.0100,-0.0100,1.0000
C01338=54.640,-112.350,44.090,0.0000,-0.0000,1.0000
C01339=50.130,-114.500,44.190,0.0000,-0.0000,1.0000
C01340=45.510,-116.410,44.190,0.0000,-0.0000,1.0000
C01341=40.810,-118.080,44.090,0.0000,-0.0000,1.0000
C01342=35.980,-119.140,43.950,0.0000,-0.0200,1.0000
C01343=31.340,-118.910,43.810,-0.0000,-0.0100,1.0000
C01344=27.650,-117.500,43.640,-0.0100,-0.0200,1.0000
C01345=25.350,-115.170,43.320,-0.0100,-0.0100,1.0000
C01346=23.490,-112.490,42.660,0.0400,0.0200,1.0000
C01347=21.680,-110.050,41.800,0.1300,0.1100,0.9900
C01348=19.520,-108.290,40.960,0.2200,0.3100,0.9300
C01349=16.290,-107.460,40.350,0.0700,0.5500,0.8300
C01350=11.150,-107.620,40.100,-0.0400,0.5800,0.8100
C01351=5.700,-108.010,40.090,-0.0300,0.5900,0.8100
C01352=0.000,-108.170,40.100,0.0000,0.5900,0.8100
C01353=0.000,-108.170,40.100,0.0000,0.5900,0.8100
C01354=-5.700,-108.010,40.090,0.0300,0.5900,0.8100
C01355=-11.150,-107.620,40.100,0.0400,0.5800,0.8100
C01356=-16.290,-107.460,40.350,-0.0700,0.5500,0.8300
C01357=-19.520,-108.290,40.960,-0.2200,0.3100,0.9300
C01358=-21.680,-110.050,41.800,-0.1300,0.1100,0.9900
C01359=-23.490,-112.490,42.660,-0.0400,0.0200,1.0000
C01360=-25.350,-115.170,43.320,0.0100,-0.0100,1.0000
C01361=-27.650,-117.500,43.640,0.0100,-0.0200,1.0000
C01362=-31.340,-118.910,43.810,0.0000,-0.0100,1.0000
C01363=-35.980,-119.140,43.950,-0.0000,-0.0200,1.0000
C01364=-40.810,-118.080,44.090,-0.0000,-0.0000,1.0000
C01365=-45.510,-116.410,44.190,-0.0000,-0.0000,1.0000
C01366=-50.130,-114.500,44.190,-0.0000,-0.0000,1.0000
C01367=-54.640,-112.350,44.090,-0.0000,-0.0000,1.0000
C01368=-58.800,-109.690,43.950,-0.0100,-0.0100,1.0000
C01369=-61.920,-106.240,43.810,-0.0100,-0.0100,1.0000
C01370=-63.530,-102.640,43.640,-0.0200,-0.0000,1.0000
C01371=-63.520,-99.360,43.320,-0.0100,0.0000,1.0000
C01372=-62.930,-96.150,42.660,0.0400,-0.0100,1.0000
C01373=-62.490,-93.150,41.800,0.1700,-0.0200,0.9900
C01374=-62.770,-90.380,40.960,0.3700,0.0700,0.9300
C01375=-64.460,-87.500,40.350,0.4300,0.3400,0.8300
C01376=-68.210,-83.980,40.100,0.3900,0.4400,0.8100
C01377=-72.340,-80.410,40.090,0.3900,0.4400,0.8100
C01378=-76.490,-76.490,40.100,0.4200,0.4200,0.8100
C01379=-80.410,-72.350,40.090,0.4400,0.3900,0.8100
C01380=-83.980,-68.210,40.100,0.4400,0.3900,0.8100
C01381=-87.500,-64.460,40.350,0.3400,0.4300,0.8300
C01382=-90.380,-62.770,40.960,0.0700,0.3700,0.9300
C01383=-93.150,-62.490,41.800,-0.0200,0.1700,0.9900
C01384=-96.150,-62.930,42.660,-0.0100,0.0400,1.0000
C01385=-99.360,-63.520,43.320,0.0000,-0.0100,1.0000
C01386=-102.640,-63.530,43.640,-0.0000,-0.0200,1.0000
C01387=-106.240,-61.920,43.810,-0.0100,-0.0100,1.0000
C01388=-109.690,-58.800,43.950,-0.0100,-0.0100,1.0000
C01389=-112.350,-54.640,44.090,-0.0000,-0.0000,1.0000
C01390=-114.500,-50.130,44.190,-0.0000,-0.0000,1.0000
C01391=-116.410,-45.510,44.190,-0.0000,-0.0000,1.0000
C01392=-118.080,-40.810,44.090,-0.0000,-0.0000,1.0000
C01393=-119.140,-35.980,43.950,-0.0200,-0.0000,1.0000
C01394=-118.910,-31.340,43.810,-0.0100,0.0000,1.0000
C01395=-117.500,-27.650,43.640,-0.0200,0.0100,1.0000
C01396=-115.170,-25.350,43.320,-0.0100,0.0100,1.0000
C01397=-112.490,-23.490,42.660,0.0200,-0.0400,1.0000
C01398=-110.050,-21.680,41.800,0.1100,-0.1300,0.9900
C01399=-108.290,-19.520,40.960,0.3100,-0.2200,0.9300
C01400=-107.460,-16.290,40.350,0.5500,-0.0700,0.8300
C01401=-107.620,-11.150,40.100,0.5800,0.0400,0.8100
C01402=-108.010,-5.700,40.090,0.5900,0.0300,0.8100
C01403=-108.170,0.000,40.100,0.5900,-0.0000,0.8100
C01404=-108.010,5.700,40.090,0.5900,-0.0300,0.8100
C01405=-107.620,11.150,40.100,0.5800,-0.0400,0.8100
C01406=-107.460,16.290,40.350,0.5500,0.0700,0.8300
C01407=-108.290,19.520,40.960,0.3100,0.2200,0.9300
C01408=-110.050,21.680,41.800,0.1100,0.1300,0.9900
C01409=-112.490,23.490,42.660,0.0200,0.0400,1.0000
C01410=-115.170,25.350,43.320,-0.0100,-0.0100,1.0000
C01411=-117.500,27.650,43.640,-0.0200,-0.0100,1.0000
C01412=-118.910,31.340,43.810,-0.0100,-0.0000,1.0000
C01413=-119.140,35.980,43.950,-0.0200,0.0000,1.0000
C01414=-118.080,40.810,44.090,-0.0000,0.0000,1.0000
C01415=-116.410,45.510,44.190,-0.0000,0.0000,1.0000
C01416=-114.500,50.130,44.190,-0.0000,0.0000,1.0000
C01417=-112.350,54.640,44.090,-0.0000,0.0000,1.0000
C01418=-109.690,58.800,43.950,-0.0100,0.0100,1.0000
C01419=-106.240,61.920,43.810,-0.0100,0.0100,1.0000
C01420=-102.640,63.530,43.640,-0.0000,0.0200,1.0000
C01421=-99.360,63.520,43.320,0.0000,0.0100,1.0000
C01422=-96.150,62.930,42.660,-0.0100,-0.0400,1.0000
C01423=-93.150,62.490,41.800,-0.0200,-0.1700,0.9900
C01424=-90.380,62.770,40.960,0.0700,-0.3700,0.9300
C01425=-87.500,64.460,40.350,0.3400,-0.4300,0.8300
C01426=-83.980,68.210,40.100,0.4400,-0.3900,0.8100
C01427=-80.410,72.340,40.090,0.4400,-0.3900,0.8100
C01428=-76.490,76.490,40.100,0.4200,-0.4200,0.8100
C01429=-72.350,80.410,40.090,0.3900,-0.4400,0.8100
C01430=-68.210,83.980,40.100,0.3900,-0.4400,0.8100
C01431=-64.460,87.500,40.350,0.4300,-0.3400,0.8300
C01432=-62.770,90.380,40.960,0.3700,-0.0700,0.9300
C01433=-62.490,93.150,41.800,0.1700,0.0200,0.9900
C01434=-62.930,96.150,42.660,0.0400,0.0100,1.0000
C01435=-63.520,99.360,43.320,-0.0100,-0.0000,1.0000
C01436=-63.530,102.640,43.640,-0.0200,0.0000,1.0000
C01437=-61.920,106.240,43.810,-0.0100,0.0100,1.0000
C01438=-58.800,109.690,43.950,-0.0100,0.0100,1.0000
C01439=-54.640,112.350,44.090,-0.0000,0.0000,1.0000
C01440=-50.130,114.500,44.190,-0.0000,0.0000,1.0000
C01441=-45.510,116.410,44.190,-0.0000,0.0000,1.0000
C01442=-40.810,118.080,44.090,-0.0000,0.0000,1.0000
C01443=-35.980,119.140,43.950,-0.0000,0.0200,1.0000
C01444=-31.340,118.910,43.810,0.0000,0.0100,1.0000
C01445=-27.650,117.500,43.640,0.0100,0.0200,1.0000
C01446=-25.350,115.170,43.320,0.0100,0.0100,1.0000
C01447=-23.490,112.490,42.660,-0.0400,-0.0200,1.0000
C01448=-21.680,110.050,41.800,-0.1300,-0.1100,0.9900
C01449=-19.520,108.290,40.960,-0.2200,-0.3100,0.9300
C01450=-16.290,107.460,40.350,-0.0700,-0.5500,0.8300
C01451=-11.150,107.620,40.100,0.0400,-0.5800,0.8100
C01452=-5.700,108.010,40.090,0.0300,-0.5900,0.8100
C01453=0.000,108.170,40.100,0.0000,-0.5900,0.8100
C01454=0.000,107.160,41.470,0.0000,-0.5900,0.8000
C01455=-5.610,107.010,41.460,0.0300,-0.5900,0.8000
C01456=-10.990,106.630,41.470,0.0400,-0.5900,0.8100
C01457=-16.110,106.500,41.740,-0.0800,-0.5500,0.8300
C01458=-19.290,107.410,42.400,-0.2200,-0.2900,0.9300
C01459=-21.410,109.300,43.300,-0.1200,-0.0900,0.9900
C01460=-23.190,111.910,44.230,-0.0300,-0.0200,1.0000
C01461=-25.020,114.790,44.940,0.0200,0.0200,1.0000
C01462=-27.290,117.310,45.290,0.0200,0.0300,1.0000
C01463=-31.010,118.870,45.480,0.0000,0.0200,1.0000
C01464=-35.720,119.190,45.630,-0.0000,0.0200,1.0000
C01465=-40.640,118.130,45.780,-0.0000,0.0000,1.0000
C01466=-45.460,116.430,45.890,-0.0000,0.0000,1.0000
C01467=-50.190,114.470,45.890,-0.0000,0.0000,1.0000
C01468=-54.800,112.270,45.780,-0.0000,0.0000,1.0000
C01469=-59.020,109.530,45.630,-0.0100,0.0100,1.0000
C01470=-62.120,105.980,45.480,-0.0200,0.0100,1.0000
C01471=-63.650,102.250,45.290,-0.0300,0.0000,1.0000
C01472=-63.470,98.860,44.940,-0.0300,-0.0000,1.0000
C01473=-62.730,95.530,44.230,0.0300,0.0100,1.0000
C01474=-62.150,92.430,43.300,0.1500,0.0200,0.9900
C01475=-62.310,89.590,42.400,0.3600,-0.0500,0.9300
C01476=-63.920,86.690,41.740,0.4400,-0.3400,0.8300
C01477=-67.620,83.170,41.470,0.3900,-0.4400,0.8100
C01478=-71.700,79.640,41.460,0.4000,-0.4400,0.8000
C01479=-75.780,75.780,41.470,0.4200,-0.4200,0.8000
C01480=-79.640,71.700,41.460,0.4400,-0.4000,0.8000
C01481=-83.170,67.620,41.470,0.4400,-0.3900,0.8100
C01482=-86.690,63.920,41.740,0.3400,-0.4400,0.8300
C01483=-89.590,62.310,42.400,0.0500,-0.3600,0.9300
C01484=-92.430,62.150,43.300,-0.0200,-0.1500,0.9900
C01485=-95.530,62.730,44.230,-0.0100,-0.0300,1.0000
C01486=-98.860,63.470,44.940,0.0000,0.0300,1.0000
C01487=-102.250,63.650,45.290,-0.0000,0.0300,1.0000
C01488=-105.980,62.120,45.480,-0.0100,0.0200,1.0000
C01489=-109.530,59.020,45.630,-0.0100,0.0100,1.0000
C01490=-112.270,54.800,45.780,-0.0000,0.0000,1.0000
C01491=-114.470,50.190,45.890,-0.0000,0.0000,1.0000
C01492=-116.430,45.460,45.890,-0.0000,0.0000,1.0000
C01493=-118.130,40.640,45.780,-0.0000,0.0000,1.0000
C01494=-119.190,35.720,45.630,-0.0200,0.0000,1.0000
C01495=-118.870,31.010,45.480,-0.0200,-0.0000,1.0000
C01496=-117.310,27.290,45.290,-0.0300,-0.0200,1.0000
C01497=-114.790,25.020,44.940,-0.0200,-0.0200,1.0000
C01498=-111.910,23.190,44.230,0.0200,0.0300,1.0000
C01499=-109.300,21.410,43.300,0.0900,0.1200,0.9900
C01500=-107.410,19.290,42.400,0.2900,0.2200,0.9300
C01501=-106.500,16.110,41.740,0.5500,0.0800,0.8300
C01502=-106.630,10.990,41.470,0.5900,-0.0400,0.8100
C01503=-107.010,5.610,41.460,0.5900,-0.0300,0.8000
C01504=-107.160,0.000,41.470,0.5900,-0.0000,0.8000
C01505=-107.010,-5.610,41.460,0.5900,0.0300,0.8000
C01506=-106.630,-10.990,41.470,0.5900,0.0400,0.8100
C01507=-106.500,-16.110,41.740,0.5500,-0.0800,0.8300
C01508=-107.410,-19.290,42.400,0.2900,-0.2200,0.9300
C01509=-109.300,-21.410,43.300,0.0900,-0.1200,0.9900
C01510=-111.910,-23.190,44.230,0.0200,-0.0300,1.0000
C01511=-114.790,-25.020,44.940,-0.0200,0.0200,1.0000
C01512=-117.310,-27.290,45.290,-0.0300,0.0200,1.0000
C01513=-118.870,-31.010,45.480,-0.0200,0.0000,1.0000
C01514=-119.190,-35.720,45.630,-0.0200,-0.0000,1.0000
C01515=-118.130,-40.640,45.780,-0.0000,-0.0000,1.0000
C01516=-116.430,-45.460,45.890,-0.0000,-0.0000,1.0000
C01517=-114.470,-50.190,45.890,-0.0000,-0.0000,1.0000
C01518=-112.270,-54.800,45.780,-0.0000,-0.0000,1.0000
C01519=-109.530,-59.020,45.630,-0.0100,-0.0100,1.0000
C01520=-105.980,-62.120,45.480,-0.0100,-0.0200,1.0000
C01521=-102.250,-63.650,45.290,-0.0000,-0.0300,1.0000
C01522=-98.860,-63.470,44.940,0.0000,-0.0300,1.0000
C01523=-95.530,-62.730,44.230,-0.0100,0.0300,1.0000
C01524=-92.430,-62.150,43.300,-0.0200,0.1500,0.9900
C01525=-89.590,-62.310,42.400,0.0500,0.3600,0.9300
C01526=-86.690,-63.920,41.740,0.3400,0.4400,0.8300
C01527=-83.170,-67.620,41.470,0.4400,0.3900,0.8100
C01528=-79.640,-71.700,41.460,0.4400,0.4000,0.8000
C01529=-75.780,-75.780,41.470,0.4200,0.4200,0.8000
C01530=-71.700,-79.640,41.460,0.4000,0.4400,0.8000
C01531=-67.620,-83.170,41.470,0.3900,0.4400,0.8100
C01532=-63.920,-86.690,41.740,0.4400,0.3400,0.8300
C01533=-62.310,-89.590,42.400,0.3600,0.0500,0.9300
C01534=-62.150,-92.430,43.300,0.1500,-0.0200,0.9900
C01535=-62.730,-95.530,44.230,0.0300,-0.0100,1.0000
C01536=-63.470,-98.860,44.940,-0.0300,0.0000,1.0000
C01537=-63.650,-102.250,45.290,-0.0300,-0.0000,1.0000
C01538=-62.120,-105.980,45.480,-0.0200,-0.0100,1.0000
C01539=-59.020,-109.530,45.630,-0.0100,-0.0100,1.0000
C01540=-54.800,-112.270,45.780,-0.0000,-0.0000,1.0000
C01541=-50.190,-114.470,45.890,-0.0000,-0.0000,1.0000
C01542=-45.460,-116.430,45.890,-0.0000,-0.0000,1.0000
C01543=-40.640,-118.130,45.780,-0.0000,-0.0000,1.0000
C01544=-35.720,-119.190,45.630,-0.0000,-0.0200,1.0000
C01545=-31.010,-118.870,45.480,0.0000,-0.0200,1.0000
C01546=-27.290,-117.310,45.290,0.0200,-0.0300,1.0000
C01547=-25.020,-114.790,44.940,0.0200,-0.0200,1.0000
C01548=-23.190,-111.910,44.230,-0.0300,0.0200,1.0000
C01549=-21.410,-109.300,43.300,-0.1200,0.0900,0.9900
C01550=-19.290,-107.410,42.400,-0.2200,0.2900,0.9300
C01551=-16.110,-106.500,41.740,-0.0800,0.5500,0.8300
C01552=-10.990,-106.630,41.470,0.0400,0.5900,0.8100
C01553=-5.610,-107.010,41.460,0.0300,0.5900,0.8000
C01554=0.000,-107.160,41.470,0.0000,0.5900,0.8000
C01555=0.000,-107.160,41.470,0.0000,0.5900,0.8000
C01556=5.610,-107.010,41.460,-0.0300,0.5900,0.8000
C01557=10.990,-106.630,41.470,-0.0400,0.5900,0.8100
C01558=16.110,-106.500,41.740,0.0800,0.5500,0.8300
C01559=19.290,-107.410,42.400,0.2200,0.2900,0.9300
C01560=21.410,-109.300,43.300,0.1200,0.0900,0.9900
C01561=23.190,-111.910,44.230,0.0300,0.0200,1.0000
C01562=25.020,-114.790,44.940,-0.0200,-0.0200,1.0000
C01563=27.290,-117.310,45.290,-0.0200,-0.0300,1.0000
C01564=31.010,-118.870,45.480,-0.0000,-0.0200,1.0000
C01565=35.720,-119.190,45.630,0.0000,-0.0200,1.0000
C01566=40.640,-118.130,45.780,0.0000,-0.0000,1.0000
C01567=45.460,-116.430,45.890,0.0000,-0.0000,1.0000
C01568=50.190,-114.470,45.890,0.0000,-0.0000,1.0000
C01569=54.800,-112.270,45.780,0.0000,-0.0000,1.0000
C01570=59.020,-109.530,45.630,0.0100,-0.0100,1.0000
C01571=62.120,-105.980,45.480,0.0200,-0.0100,1.0000
C01572=63.650,-102.250,45.290,0.0300,-0.0000,1.0000
C01573=63.470,-98.860,44.940,0.0300,0.0000,1.0000
C01574=62.730,-95.530,44.230,-0.0300,-0.0100,1.0000
C01575=62.150,-92.430,43.300,-0.1500,-0.0200,0.9900
C01576=62.310,-89.590,42.400,-0.3600,0.0500,0.9300
C01577=63.920,-86.690,41.740,-0.4400,0.3400,0.8300
C01578=67.620,-83.170,41.470,-0.3900,0.4400,0.8100
C01579=71.700,-79.640,41.460,-0.4000,0.4400,0.8000
C01580=75.780,-75.780,41.470,-0.4200,0.4200,0.8000
C01581=79.640,-71.700,41.460,-0.4400,0.4000,0.8000
C01582=83.170,-67.620,41.470,-0.4400,0.3900,0.8100
C01583=86.690,-63.920,41.740,-0.3400,0.4400,0.8300
C01584=89.590,-62.310,42.400,-0.0500,0.3600,0.9300
C01585=92.430,-62.150,43.300,0.0200,0.1500,0.9900
C01586=95.530,-62.730,44.230,0.0100,0.0300,1.0000
C01587=98.860,-63.470,44.940,-0.0000,-0.0300,1.0000
C01588=102.250,-63.650,45.290,0.0000,-0.0300,1.0000
C01589=105.980,-62.120,45.480,0.0100,-0.0200,1.0000
C01590=109.530,-59.020,45.630,0.0100,-0.0100,1.0000
C01591=112.270,-54.800,45.780,0.0000,-0.0000,1.0000
C01592=114.470,-50.190,45.890,0.0000,-0.0000,1.0000
C01593=116.430,-45.460,45.890,0.0000,-0.0000,1.0000
C01594=118.130,-40.640,45.780,0.0000,-0.0000,1.0000
C01595=119.190,-35.720,45.630,0.0200,-0.0000,1.0000
C01596=118.870,-31.010,45.480,0.0200,0.0000,1.0000
C01597=117.310,-27.290,45.290,0.0300,0.0200,1.0000
C01598=114.790,-25.020,44.940,0.0200,0.0200,1.0000
C01599=111.910,-23.190,44.230,-0.0200,-0.0300,1.0000
C01600=109.300,-21.410,43.300,-0.0900,-0.1200,0.9900
C01601=107.410,-19.290,42.400,-0.2900,-0.2200,0.9300
C01602=106.500,-16.110,41.740,-0.5500,-0.0800,0.8300
C01603=106.630,-10.990,41.470,-0.5900,0.0400,0.8100
C01604=107.010,-5.610,41.460,-0.5900,0.0300,0.8000
C01605=107.160,0.000,41.470,-0.5900,0.0000,0.8000
C01606=107.010,5.610,41.460,-0.5900,-0.0300,0.8000
C01607=106.630,10.990,41.470,-0.5900,-0.0400,0.8100
C01608=106.500,16.110,41.740,-0.5500,0.0800,0.8300
C01609=107.410,19.290,42.400,-0.2900,0.2200,0.9300
C01610=109.300,21.410,43.300,-0.0900,0.1200,0.9900
C01611=111.910,23.190,44.230,-0.0200,0.0300,1.0000
C01612=114.790,25.020,44.940,0.0200,-0.0200,1.0000
C01613=117.310,27.290,45.290,0.0300,-0.0200,1.0000
C01614=118.870,31.010,45.480,0.0200,-0.0000,1.0000
C01615=119.190,35.720,45.630,0.0200,0.0000,1.0000
C01616=118.130,40.640,45.780,0.0000,0.0000,1.0000
C01617=116.430,45.460,45.890,0.0000,0.0000,1.0000
C01618=114.470,50.190,45.890,0.0000,0.0000,1.0000
C01619=112.270,54.800,45.780,0.0000,0.0000,1.0000
C01620=109.530,59.020,45.630,0.0100,0.0100,1.0000
C01621=105.980,62.120,45.480,0.0100,0.0200,1.0000
C01622=102.250,63.650,45.290,0.0000,0.0300,1.0000
C01623=98.860,63.470,44.940,-0.0000,0.0300,1.0000
C01624=95.530,62.730,44.230,0.0100,-0.0300,1.0000
C01625=92.430,62.150,43.300,0.0200,-0.1500,0.9900
C01626=89.590,62.310,42.400,-0.0500,-0.3600,0.9300
C01627=86.690,63.920,41.740,-0.3400,-0.4400,0.8300
C01628=83.170,67.620,41.470,-0.4400,-0.3900,0.8100
C01629=79.640,71.700,41.460,-0.4400,-0.4000,0.8000
C01630=75.780,75.780,41.470,-0.4200,-0.4200,0.8000
C01631=71.700,79.640,41.460,-0.4000,-0.4400,0.8000
C01632=67.620,83.170,41.470,-0.3900,-0.4400,0.8100
C01633=63.920,86.690,41.740,-0.4400,-0.3400,0.8300
C01634=62.310,89.590,42.400,-0.3600,-0.0500,0.9300
C01635=62.150,92.430,43.300,-0.1500,0.0200,0.9900
C01636=62.730,95.530,44.230,-0.0300,0.0100,1.0000
C01637=63.470,98.860,44.940,0.0300,-0.0000,1.0000
C01638=63.650,102.250,45.290,0.0300,0.0000,1.0000
C01639=62.120,105.980,45.480,0.0200,0.0100,1.0000
C01640=59.020,109.530,45.630,0.0100,0.0100,1.0000
C01641=54.800,112.270,45.780,0.0000,0.0000,1.0000
C01642=50.190,114.470,45.890,0.0000,0.0000,1.0000
C01643=45.460,116.430,45.890,0.0000,0.0000,1.0000
C01644=40.640,118.130,45.780,0.0000,0.0000,1.0000
C01645=35.720,119.190,45.630,0.0000,0.0200,1.0000
C01646=31.010,118.870,45.480,-0.0000,0.0200,1.0000
C01647=27.290,117.310,45.290,-0.0200,0.0300,1.0000
C01648=25.020,114.790,44.940,-0.0200,0.0200,1.0000
C01649=23.190,111.910,44.230,0.0300,-0.0200,1.0000
C01650=21.410,109.300,43.300,0.1200,-0.0900,0.9900
C01651=19.290,107.410,42.400,0.2200,-0.2900,0.9300
C01652=16.110,106.500,41.740,0.0800,-0.5500,0.8300
C01653=10.990,106.630,41.470,-0.0400,-0.5900,0.8100
C01654=5.610,107.010,41.460,-0.0300,-0.5900,0.8000
C01655=0.000,107.160,41.470,0.0000,-0.5900,0.8000
C01656=0.000,106.150,42.830,0.0000,-0.6000,0.8000
C01657=5.520,106.000,42.820,-0.0300,-0.6000,0.8000
C01658=10.840,105.620,42.840,-0.0300,-0.6000,0.8000
C01659=15.910,105.520,43.120,0.0900,-0.5500,0.8300
C01660=19.050,106.520,43.820,0.2200,-0.2700,0.9400
C01661=21.140,108.540,44.790,0.1100,-0.0800,0.9900
C01662=22.890,111.320,45.790,0.0100,-0.0100,1.0000
C01663=24.690,114.400,46.560,-0.0300,0.0200,1.0000
C01664=26.930,117.110,46.940,-0.0300,0.0300,1.0000
C01665=30.670,118.820,47.140,-0.0100,0.0200,1.0000
C01666=35.450,119.240,47.310,0.0000,0.0200,1.0000
C01667=40.470,118.190,47.470,0.0000,0.0000,1.0000
C01668=45.400,116.450,47.590,0.0000,0.0000,1.0000
C01669=50.240,114.450,47.590,0.0000,0.0000,1.0000
C01670=54.960,112.190,47.470,0.0000,0.0000,1.0000
C01671=59.250,109.380,47.310,0.0100,0.0100,1.0000
C01672=62.340,105.710,47.140,0.0200,0.0100,1.0000
C01673=63.760,101.850,46.940,0.0400,0.0000,1.0000
C01674=63.430,98.350,46.560,0.0400,-0.0100,1.0000
C01675=62.520,94.900,45.790,-0.0200,0.0000,1.0000
C01676=61.800,91.700,44.790,-0.1300,0.0300,0.9900
C01677=61.850,88.790,43.820,-0.3500,-0.0300,0.9400
C01678=63.360,85.870,43.120,-0.4500,-0.3300,0.8300
C01679=67.020,82.350,42.840,-0.4000,-0.4500,0.8000
C01680=71.050,78.860,42.820,-0.4000,-0.4500,0.8000
C01681=75.060,75.060,42.830,-0.4200,-0.4200,0.8000
C01682=78.860,71.050,42.820,-0.4500,-0.4000,0.8000
C01683=82.350,67.020,42.840,-0.4500,-0.4000,0.8000
C01684=85.870,63.360,43.120,-0.3300,-0.4500,0.8300
C01685=88.790,61.850,43.820,-0.0300,-0.3500,0.9400
C01686=91.700,61.800,44.790,0.0300,-0.1300,0.9900
C01687=94.900,62.520,45.790,0.0000,-0.0200,1.0000
C01688=98.350,63.430,46.560,-0.0100,0.0400,1.0000
C01689=101.850,63.760,46.940,0.0000,0.0400,1.0000
C01690=105.710,62.340,47.140,0.0100,0.0200,1.0000
C01691=109.380,59.250,47.310,0.0100,0.0100,1.0000
C01692=112.190,54.960,47.470,0.0000,0.0000,1.0000
C01693=114.450,50.240,47.590,0.0000,0.0000,1.0000
C01694=116.450,45.400,47.590,0.0000,0.0000,1.0000
C01695=118.190,40.470,47.470,0.0000,0.0000,1.0000
C01696=119.240,35.450,47.310,0.0200,0.0000,1.0000
C01697=118.820,30.670,47.140,0.0200,-0.0100,1.0000
C01698=117.110,26.930,46.940,0.0300,-0.0300,1.0000
C01699=114.400,24.690,46.560,0.0200,-0.0300,1.0000
C01700=111.320,22.890,45.790,-0.0100,0.0100,1.0000
C01701=108.540,21.140,44.790,-0.0800,0.1100,0.9900
C01702=106.520,19.050,43.820,-0.2700,0.2200,0.9400
C01703=105.520,15.910,43.120,-0.5500,0.0900,0.8300
C01704=105.620,10.840,42.840,-0.6000,-0.0300,0.8000
C01705=106.000,5.520,42.820,-0.6000,-0.0300,0.8000
C01706=106.150,0.000,42.830,-0.6000,0.0000,0.8000
C01707=106.000,-5.520,42.820,-0.6000,0.0300,0.8000
C01708=105.620,-10.840,42.840,-0.6000,0.0300,0.8000
C01709=105.530,-15.910,43.120,-0.5500,-0.0900,0.8300
C01710=106.520,-19.050,43.820,-0.2700,-0.2200,0.9400
C01711=108.540,-21.140,44.790,-0.0800,-0.1100,0.9900
C01712=111.320,-22.890,45.790,-0.0100,-0.0100,1.0000
C01713=114.400,-24.690,46.560,0.0200,0.0300,1.0000
C01714=117.110,-26.930,46.940,0.0300,0.0300,1.0000
C01715=118.820,-30.670,47.140,0.0200,0.0100,1.0000
C01716=119.240,-35.450,47.310,0.0200,-0.0000,1.0000
C01717=118.190,-40.470,47.470,0.0000,-0.0000,1.0000
C01718=116.450,-45.400,47.590,0.0000,-0.0000,1.0000
C01719=114.450,-50.240,47.590,0.0000,-0.0000,1.0000
C01720=112.190,-54.960,47.470,0.0000,-0.0000,1.0000
C01721=109.380,-59.250,47.310,0.0100,-0.0100,1.0000
C01722=105.710,-62.340,47.140,0.0100,-0.0200,1.0000
C01723=101.850,-63.760,46.940,0.0000,-0.0400,1.0000
C01724=98.350,-63.430,46.560,-0.0100,-0.0400,1.0000
C01725=94.900,-62.520,45.790,0.0000,0.0200,1.0000
C01726=91.700,-61.800,44.790,0.0300,0.1300,0.9900
C01727=88.790,-61.850,43.820,-0.0300,0.3500,0.9400
C01728=85.870,-63.360,43.120,-0.3300,0.4500,0.8300
C01729=82.350,-67.020,42.840,-0.4500,0.4000,0.8000
C01730=78.860,-71.050,42.820,-0.4500,0.4000,0.8000
C01731=75.060,-75.060,42.830,-0.4200,0.4200,0.8000
C01732=71.050,-78.860,42.820,-0.4000,0.4500,0.8000
C01733=67.020,-82.350,42.840,-0.4000,0.4500,0.8000
C01734=63.360,-85.870,43.120,-0.4500,0.3300,0.8300
C01735=61.850,-88.790,43.820,-0.3500,0.0300,0.9400
C01736=61.800,-91.700,44.790,-0.1300,-0.0300,0.9900
C01737=62.520,-94.900,45.790,-0.0200,-0.0000,1.0000
C01738=63.430,-98.350,46.560,0.0400,0.0100,1.0000
C01739=63.760,-101.850,46.940,0.0400,-0.0000,1.0000
C01740=62.340,-105.710,47.140,0.0200,-0.0100,1.0000
C01741=59.250,-109.380,47.310,0.0100,-0.0100,1.0000
C01742=54.960,-112.190,47.470,0.0000,-0.0000,1.0000
C01743=50.240,-114.450,47.590,0.0000,-0.0000,1.0000
C01744=45.400,-116.450,47.590,0.0000,-0.0000,1.0000
C01745=40.470,-118.190,47.470,0.0000,-0.0000,1.0000
C01746=35.450,-119.240,47.310,0.0000,-0.0200,1.0000
C01747=30.670,-118.820,47.140,-0.0100,-0.0200,1.0000
C01748=26.930,-117.110,46.940,-0.0300,-0.0300,1.0000
C01749=24.690,-114.400,46.560,-0.0300,-0.0200,1.0000
C01750=22.890,-111.320,45.790,0.0100,0.0100,1.0000
C01751=21.140,-108.540,44.790,0.1100,0.0800,0.9900
C01752=19.050,-106.520,43.820,0.2200,0.2700,0.9400
C01753=15.910,-105.520,43.120,0.0900,0.5500,0.8300
C01754=10.840,-105.620,42.840,-0.0300,0.6000,0.8000
C01755=5.520,-106.000,42.820,-0.0300,0.6000,0.8000
C01756=0.000,-106.150,42.830,0.0000,0.6000,0.8000
C01757=0.000,-106.150,42.830,0.0000,0.6000,0.8000
C01758=-5.520,-106.000,42.820,0.0300,0.6000,0.8000
C01759=-10.840,-105.620,42.840,0.0300,0.6000,0.8000
C01760=-15.910,-105.530,43.120,-0.0900,0.5500,0.8300
C01761=-19.050,-106.520,43.820,-0.2200,0.2700,0.9400
C01762=-21.140,-108.540,44.790,-0.1100,0.0800,0.9900
C01763=-22.890,-111.320,45.790,-0.0100,0.0100,1.0000
C01764=-24.690,-114.400,46.560,0.0300,-0.0200,1.0000
C01765=-26.930,-117.110,46.940,0.0300,-0.0300,1.0000
C01766=-30.670,-118.820,47.140,0.0100,-0.0200,1.0000
C01767=-35.450,-119.240,47.310,-0.0000,-0.0200,1.0000
C01768=-40.470,-118.190,47.470,-0.0000,-0.0000,1.0000
C01769=-45.400,-116.450,47.590,-0.0000,-0.0000,1.0000
C01770=-50.240,-114.450,47.590,-0.0000,-0.0000,1.0000
C01771=-54.960,-112.190,47.470,-0.0000,-0.0000,1.0000
C01772=-59.250,-109.380,47.310,-0.0100,-0.0100,1.0000
C01773=-62.340,-105.710,47.140,-0.0200,-0.0100,1.0000
C01774=-63.760,-101.850,46.940,-0.0400,-0.0000,1.0000
C01775=-63.430,-98.350,46.560,-0.0400,0.0100,1.0000
C01776=-62.520,-94.900,45.790,0.0200,-0.0000,1.0000
C01777=-61.800,-91.700,44.790,0.1300,-0.0300,0.9900
C01778=-61.850,-88.790,43.820,0.3500,0.0300,0.9400
C01779=-63.360,-85.870,43.120,0.4500,0.3300,0.8300
C01780=-67.020,-82.350,42.840,0.4000,0.4500,0.8000
C01781=-71.050,-78.860,42.820,0.4000,0.4500,0.8000
C01782=-75.060,-75.060,42.830,0.4200,0.4200,0.8000
C01783=-78.860,-71.050,42.820,0.4500,0.4000,0.8000
C01784=-82.350,-67.020,42.840,0.4500,0.4000,0.8000
C01785=-85.870,-63.360,43.120,0.3300,0.4500,0.8300
C01786=-88.790,-61.850,43.820,0.0300,0.3500,0.9400
C01787=-91.700,-61.800,44.790,-0.0300,0.1300,0.9900
C01788=-94.900,-62.520,45.790,-0.0000,0.0200,1.0000
C01789=-98.350,-63.430,46.560,0.0100,-0.0400,1.0000
C01790=-101.850,-63.760,46.940,-0.0000,-0.0400,1.0000
C01791=-105.710,-62.340,47.140,-0.0100,-0.0200,1.0000
C01792=-109.380,-59.250,47.310,-0.0100,-0.0100,1.0000
C01793=-112.190,-54.960,47.470,-0.0000,-0.0000,1.0000
C01794=-114.450,-50.240,47.590,-0.0000,-0.0000,1.0000
C01795=-116.450,-45.400,47.590,-0.0000,-0.0000,1.0000
C01796=-118.190,-40.470,47.470,-0.0000,-0.0000,1.0000
C01797=-119.240,-35.450,47.310,-0.0200,-0.0000,1.0000
C01798=-118.820,-30.670,47.140,-0.0200,0.0100,1.0000
C01799=-117.110,-26.930,46.940,-0.0300,0.0300,1.0000
C01800=-114.400,-24.690,46.560,-0.0200,0.0300,1.0000
C01801=-111.320,-22.890,45.790,0.0100,-0.0100,1.0000
C01802=-108.540,-21.140,44.790,0.0800,-0.1100,0.9900
C01803=-106.520,-19.050,43.820,0.2700,-0.2200,0.9400
C01804=-105.520,-15.910,43.120,0.5500,-0.0900,0.8300
C01805=-105.620,-10.840,42.840,0.6000,0.0300,0.8000
C01806=-106.000,-5.520,42.820,0.6000,0.0300,0.8000
C01807=-106.150,0.000,42.830,0.6000,-0.0000,0.8000
C01808=-106.000,5.520,42.820,0.6000,-0.0300,0.8000
C01809=-105.620,10.840,42.840,0.6000,-0.0300,0.8000
C01810=-105.530,15.910,43.120,0.5500,0.0900,0.8300
C01811=-106.520,19.050,43.820,0.2700,0.2200,0.9400
C01812=-108.540,21.140,44.790,0.0800,0.1100,0.9900
C01813=-111.320,22.890,45.790,0.0100,0.0100,1.0000
C01814=-114.400,24.690,46.560,-0.0200,-0.0300,1.0000
C01815=-117.110,26.930,46.940,-0.0300,-0.0300,1.0000
C01816=-118.820,30.670,47.140,-0.0200,-0.0100,1.0000
C01817=-119.240,35.450,47.310,-0.0200,0.0000,1.0000
C01818=-118.190,40.470,47.470,-0.0000,0.0000,1.0000
C01819=-116.450,45.400,47.590,-0.0000,0.0000,1.0000
C01820=-114.450,50.240,47.590,-0.0000,0.0000,1.0000
C01821=-112.190,54.960,47.470,-0.0000,0.0000,1.0000
C01822=-109.380,59.250,47.310,-0.0100,0.0100,1.0000
C01823=-105.710,62.340,47.140,-0.0100,0.0200,1.0000
C01824=-101.850,63.760,46.940,-0.0000,0.0400,1.0000
C01825=-98.350,63.430,46.560,0.0100,0.0400,1.0000
C01826=-94.900,62.520,45.790,-0.0000,-0.0200,1.0000
C01827=-91.700,61.800,44.790,-0.0300,-0.1300,0.9900
C01828=-88.790,61.850,43.820,0.0300,-0.3500,0.9400
C01829=-85.870,63.360,43.120,0.3300,-0.4500,0.8300
C01830=-82.350,67.020,42.840,0.4500,-0.4000,0.8000
C01831=-78.860,71.050,42.820,0.4500,-0.4000,0.8000
C01832=-75.060,75.060,42.830,0.4200,-0.4200,0.8000
C01833=-71.050,78.860,42.820,0.4000,-0.4500,0.8000
C01834=-67.020,82.350,42.840,0.4000,-0.4500,0.8000
C01835=-63.360,85.870,43.120,0.4500,-0.3300,0.8300
C01836=-61.850,88.790,43.820,0.3500,-0.0300,0.9400
C01837=-61.800,91.700,44.790,0.1300,0.0300,0.9900
C01838=-62.520,94.900,45.790,0.0200,0.0000,1.0000
C01839=-63.430,98.350,46.560,-0.0400,-0.0100,1.0000
C01840=-63.760,101.850,46.940,-0.0400,0.0000,1.0000
C01841=-62.340,105.710,47.140,-0.0200,0.0100,1.0000
C01842=-59.250,109.380,47.310,-0.0100,0.0100,1.0000
C01843=-54.960,112.190,47.470,-0.0000,0.0000,1.0000
C01844=-50.240,114.450,47.590,-0.0000,0.0000,1.0000
C01845=-45.400,116.450,47.590,-0.0000,0.0000,1.0000
C01846=-40.470,118.190,47.470,-0.0000,0.0000,1.0000
C01847=-35.450,119.240,47.310,-0.0000,0.0200,1.0000
C01848=-30.670,118.820,47.140,0.0100,0.0200,1.0000
C01849=-26.930,117.110,46.940,0.0300,0.0300,1.0000
C01850=-24.690,114.400,46.560,0.0300,0.0200,1.0000
C01851=-22.890,111.320,45.790,-0.0100,-0.0100,1.0000
C01852=-21.140,108.540,44.790,-0.1100,-0.0800,0.9900
C01853=-19.050,106.520,43.820,-0.2200,-0.2700,0.9400
C01854=-15.910,105.530,43.120,-0.0900,-0.5500,0.8300
C01855=-10.840,105.620,42.840,0.0300,-0.6000,0.8000
C01856=-5.520,106.000,42.820,0.0300,-0.6000,0.8000
C01857=0.000,106.150,42.830,0.0000,-0.6000,0.8000
C01858=0.000,105.130,44.190,0.0000,-0.6000,0.8000
C01859=-5.420,104.980,44.180,0.0300,-0.6000,0.8000
C01860=-10.680,104.610,44.190,0.0300,-0.6000,0.8000
C01861=-15.720,104.550,44.490,-0.1000,-0.5500,0.8300
C01862=-18.820,105.620,45.250,-0.2300,-0.2500,0.9400
C01863=-20.860,107.770,46.290,-0.1000,-0.0700,0.9900
C01864=-22.590,110.720,47.350,-0.0000,-0.0000,1.0000
C01865=-24.360,114.000,48.180,0.0400,0.0300,1.0000
C01866=-26.570,116.910,48.590,0.0300,0.0400,1.0000
C01867=-30.320,118.780,48.810,0.0100,0.0300,1.0000
C01868=-35.170,119.290,48.990,-0.0000,0.0200,1.0000
C01869=-40.300,118.250,49.160,-0.0000,0.0000,1.0000
C01870=-45.340,116.480,49.280,-0.0000,0.0000,1.0000
C01871=-50.300,114.420,49.280,-0.0000,0.0000,1.0000
C01872=-55.120,112.110,49.160,-0.0000,0.0000,1.0000
C01873=-59.480,109.220,48.990,-0.0100,0.0200,1.0000
C01874=-62.550,105.430,48.810,-0.0300,0.0200,1.0000
C01875=-63.880,101.460,48.590,-0.0500,0.0000,1.0000
C01876=-63.390,97.840,48.180,-0.0500,-0.0100,1.0000
C01877=-62.320,94.260,47.350,0.0000,0.0000,1.0000
C01878=-61.450,90.960,46.290,0.1200,0.0300,0.9900
C01879=-61.380,87.990,45.250,0.3400,-0.0200,0.9400
C01880=-62.810,85.040,44.490,0.4600,-0.3200,0.8300
C01881=-66.420,81.530,44.190,0.4000,-0.4500,0.8000
C01882=-70.400,78.070,44.180,0.4000,-0.4500,0.8000
C01883=-74.330,74.330,44.190,0.4300,-0.4300,0.8000
C01884=-78.070,70.400,44.180,0.4500,-0.4000,0.8000
C01885=-81.530,66.420,44.190,0.4500,-0.4000,0.8000
C01886=-85.040,62.810,44.490,0.3200,-0.4600,0.8300
C01887=-87.990,61.380,45.250,0.0200,-0.3400,0.9400
C01888=-90.960,61.450,46.290,-0.0300,-0.1200,0.9900
C01889=-94.260,62.320,47.350,-0.0000,-0.0000,1.0000
C01890=-97.840,63.390,48.180,0.0100,0.0500,1.0000
C01891=-101.460,63.880,48.590,-0.0000,0.0500,1.0000
C01892=-105.430,62.550,48.810,-0.0200,0.0300,1.0000
C01893=-109.220,59.480,48.990,-0.0200,0.0100,1.0000
C01894=-112.110,55.120,49.160,-0.0000,0.0000,1.0000
C01895=-114.420,50.300,49.280,-0.0000,0.0000,1.0000
C01896=-116.480,45.340,49.280,-0.0000,0.0000,1.0000
C01897=-118.250,40.300,49.160,-0.0000,0.0000,1.0000
C01898=-119.290,35.170,48.990,-0.0200,0.0000,1.0000
C01899=-118.780,30.320,48.810,-0.0300,-0.0100,1.0000
C01900=-116.910,26.570,48.590,-0.0400,-0.0300,1.0000
C01901=-114.000,24.360,48.180,-0.0300,-0.0400,1.0000
C01902=-110.720,22.590,47.350,0.0000,0.0000,1.0000
C01903=-107.770,20.860,46.290,0.0700,0.1000,0.9900
C01904=-105.620,18.820,45.250,0.2500,0.2300,0.9400
C01905=-104.550,15.720,44.490,0.5500,0.1000,0.8300
C01906=-104.610,10.680,44.190,0.6000,-0.0300,0.8000
C01907=-104.980,5.420,44.180,0.6000,-0.0300,0.8000
C01908=-105.130,0.000,44.190,0.6000,-0.0000,0.8000
C01909=-104.980,-5.420,44.180,0.6000,0.0300,0.8000
C01910=-104.610,-10.680,44.190,0.6000,0.0300,0.8000
C01911=-104.550,-15.720,44.490,0.5500,-0.1000,0.8300
C01912=-105.620,-18.820,45.250,0.2500,-0.2300,0.9400
C01913=-107.770,-20.860,46.290,0.0700,-0.1000,0.9900
C01914=-110.720,-22.590,47.350,0.0000,-0.0000,1.0000
C01915=-114.000,-24.360,48.180,-0.0300,0.0400,1.0000
C01916=-116.910,-26.570,48.590,-0.0400,0.0300,1.0000
C01917=-118.780,-30.320,48.810,-0.0300,0.0100,1.0000
C01918=-119.290,-35.170,48.990,-0.0200,-0.0000,1.0000
C01919=-118.250,-40.300,49.160,-0.0000,-0.0000,1.0000
C01920=-116.480,-45.340,49.280,-0.0000,-0.0000,1.0000
C01921=-114.420,-50.300,49.280,-0.0000,-0.0000,1.0000
C01922=-112.110,-55.120,49.160,-0.0000,-0.0000,1.0000
C01923=-109.220,-59.480,48.990,-0.0200,-0.0100,1.0000
C01924=-105.430,-62.550,48.810,-0.0200,-0.0300,1.0000
C01925=-101.460,-63.880,48.590,-0.0000,-0.0500,1.0000
C01926=-97.840,-63.390,48.180,0.0100,-0.0500,1.0000
C01927=-94.260,-62.320,47.350,-0.0000,0.0000,1.0000
C01928=-90.960,-61.450,46.290,-0.0300,0.1200,0.9900
